// TIA Portal V19 export
FUNCTION "TRANSFER SUBOUTPUT" : Void   // FC13, LAD
{ S7_Optimized_Access := 'TRUE' }
// stored: SetENOAutomatically false
BEGIN

REGION Network 1: SYRUP MFG VESSEL BOTTOM STERROR RUN
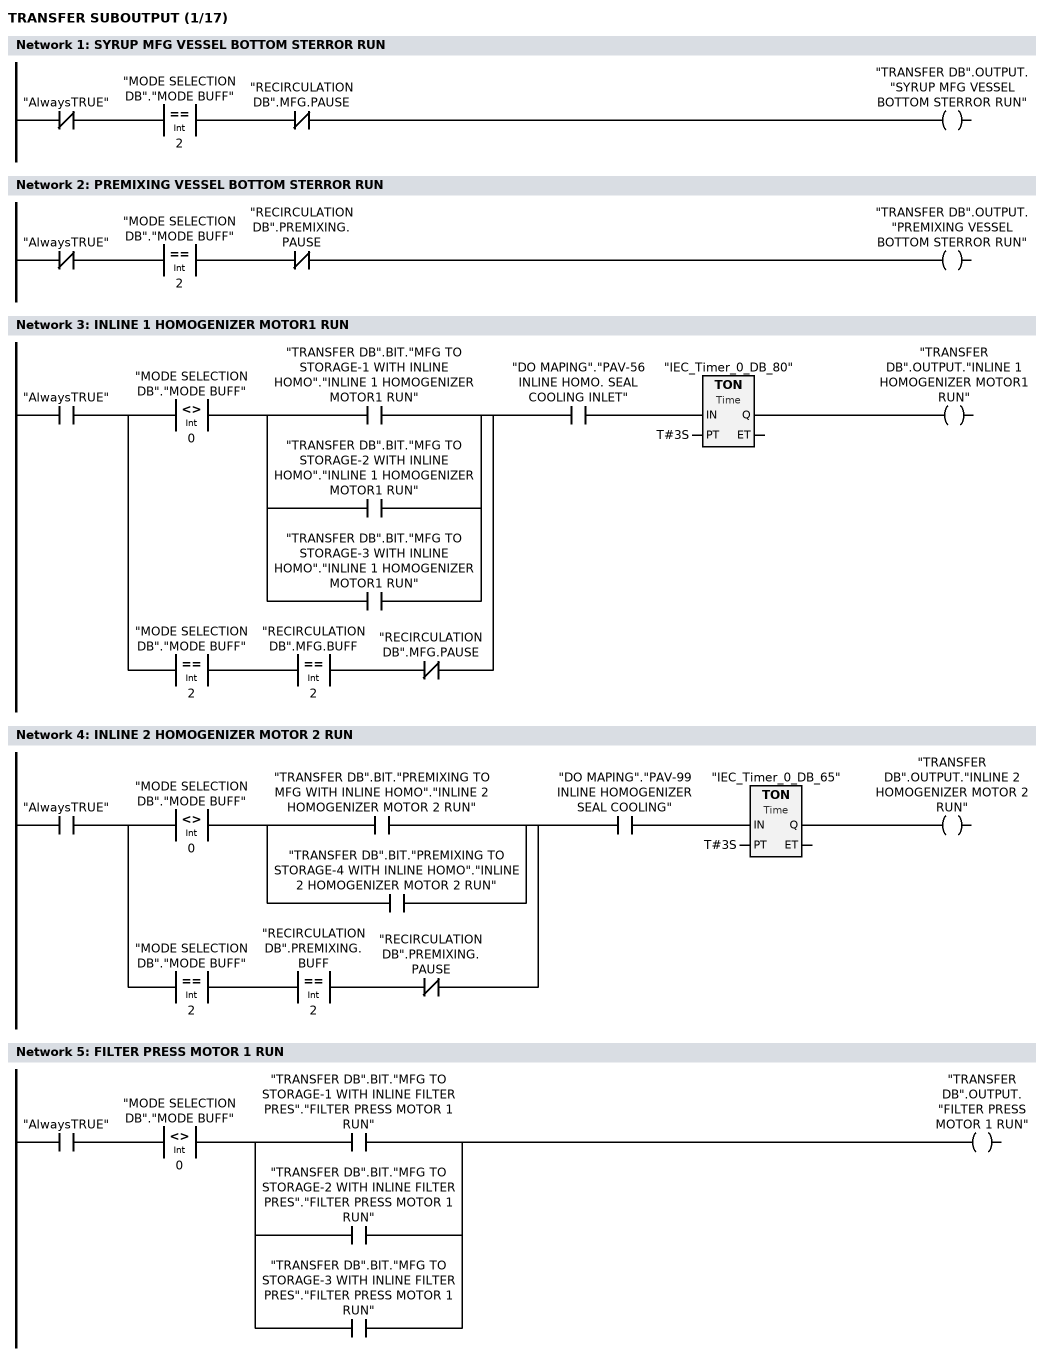
   RUNG wire#powerrail
      I_Contact( "AlwaysTRUE" )
      { S7_Templates := "SrcType := Int" } EQ_Contact(in1 := "MODE SELECTION DB"."MODE BUFF", in2 := 2)
      I_Contact( "RECIRCULATION DB".MFG.PAUSE )
      Coil( "TRANSFER DB".OUTPUT."SYRUP MFG VESSEL BOTTOM STERROR RUN" )
   END_RUNG
   // the same network as SCL:
   "TRANSFER DB".OUTPUT."SYRUP MFG VESSEL BOTTOM STERROR RUN" := NOT "AlwaysTRUE" AND ("MODE SELECTION DB"."MODE BUFF" = 2) AND NOT "RECIRCULATION DB".MFG.PAUSE;
END_REGION

REGION Network 2: PREMIXING VESSEL BOTTOM STERROR RUN
   RUNG wire#powerrail
      I_Contact( "AlwaysTRUE" )
      { S7_Templates := "SrcType := Int" } EQ_Contact(in1 := "MODE SELECTION DB"."MODE BUFF", in2 := 2)
      I_Contact( "RECIRCULATION DB".PREMIXING.PAUSE )
      Coil( "TRANSFER DB".OUTPUT."PREMIXING VESSEL BOTTOM STERROR RUN" )
   END_RUNG
   // the same network as SCL:
   "TRANSFER DB".OUTPUT."PREMIXING VESSEL BOTTOM STERROR RUN" := NOT "AlwaysTRUE" AND ("MODE SELECTION DB"."MODE BUFF" = 2) AND NOT "RECIRCULATION DB".PREMIXING.PAUSE;
END_REGION

REGION Network 3: INLINE 1 HOMOGENIZER MOTOR1 RUN
   RUNG wire#powerrail
      Contact( "AlwaysTRUE" )
      wire#w1
      { S7_Templates := "SrcType := Int" } NE_Contact(in1 := "MODE SELECTION DB"."MODE BUFF", in2 := 0)
      wire#w2
      Contact( "TRANSFER DB".BIT."MFG TO STORAGE-1 WITH INLINE HOMO"."INLINE 1 HOMOGENIZER MOTOR1 RUN" )
      wire#w3
      Contact( "DO MAPING"."PAV-56 INLINE HOMO. SEAL COOLING INLET" )
      { S7_Templates := "time_type := Time" } "IEC_Timer_0_DB_80".TON(pt := T#3S, et =>)
      Coil( "TRANSFER DB".OUTPUT."INLINE 1 HOMOGENIZER MOTOR1 RUN" )
   END_RUNG
   RUNG wire#w2
      Contact( "TRANSFER DB".BIT."MFG TO STORAGE-2 WITH INLINE HOMO"."INLINE 1 HOMOGENIZER MOTOR1 RUN" )
   END_RUNG wire#w3
   RUNG wire#w2
      Contact( "TRANSFER DB".BIT."MFG TO STORAGE-3 WITH INLINE HOMO"."INLINE 1 HOMOGENIZER MOTOR1 RUN" )
   END_RUNG wire#w3
   RUNG wire#w1
      { S7_Templates := "SrcType := Int" } EQ_Contact(in1 := "MODE SELECTION DB"."MODE BUFF", in2 := 2)
      { S7_Templates := "SrcType := Int" } EQ_Contact(in1 := "RECIRCULATION DB".MFG.BUFF, in2 := 2)
      I_Contact( "RECIRCULATION DB".MFG.PAUSE )
   END_RUNG wire#w3
   // the same network as SCL:
   "IEC_Timer_0_DB_80".TON(IN := "AlwaysTRUE" AND ((("MODE SELECTION DB"."MODE BUFF" <> 0) AND ("TRANSFER DB".BIT."MFG TO STORAGE-1 WITH INLINE HOMO"."INLINE 1 HOMOGENIZER MOTOR1 RUN" OR "TRANSFER DB".BIT."MFG TO STORAGE-2 WITH INLINE HOMO"."INLINE 1 HOMOGENIZER MOTOR1 RUN" OR "TRANSFER DB".BIT."MFG TO STORAGE-3 WITH INLINE HOMO"."INLINE 1 HOMOGENIZER MOTOR1 RUN")) OR (("MODE SELECTION DB"."MODE BUFF" = 2) AND ("RECIRCULATION DB".MFG.BUFF = 2) AND NOT "RECIRCULATION DB".MFG.PAUSE)) AND "DO MAPING"."PAV-56 INLINE HOMO. SEAL COOLING INLET",
                           PT := T#3S);
   "TRANSFER DB".OUTPUT."INLINE 1 HOMOGENIZER MOTOR1 RUN" := "IEC_Timer_0_DB_80".Q;
END_REGION

REGION Network 4: INLINE 2 HOMOGENIZER MOTOR 2 RUN
   RUNG wire#powerrail
      Contact( "AlwaysTRUE" )
      wire#w1
      { S7_Templates := "SrcType := Int" } NE_Contact(in1 := "MODE SELECTION DB"."MODE BUFF", in2 := 0)
      wire#w2
      Contact( "TRANSFER DB".BIT."PREMIXING TO MFG WITH INLINE HOMO"."INLINE 2 HOMOGENIZER MOTOR 2 RUN" )
      wire#w3
      Contact( "DO MAPING"."PAV-99 INLINE HOMOGENIZER SEAL COOLING" )
      { S7_Templates := "time_type := Time" } "IEC_Timer_0_DB_65".TON(pt := T#3S, et =>)
      Coil( "TRANSFER DB".OUTPUT."INLINE 2 HOMOGENIZER MOTOR 2 RUN" )
   END_RUNG
   RUNG wire#w2
      Contact( "TRANSFER DB".BIT."PREMIXING TO STORAGE-4 WITH INLINE HOMO"."INLINE 2 HOMOGENIZER MOTOR 2 RUN" )
   END_RUNG wire#w3
   RUNG wire#w1
      { S7_Templates := "SrcType := Int" } EQ_Contact(in1 := "MODE SELECTION DB"."MODE BUFF", in2 := 2)
      { S7_Templates := "SrcType := Int" } EQ_Contact(in1 := "RECIRCULATION DB".PREMIXING.BUFF, in2 := 2)
      I_Contact( "RECIRCULATION DB".PREMIXING.PAUSE )
   END_RUNG wire#w3
   // the same network as SCL:
   "IEC_Timer_0_DB_65".TON(IN := "AlwaysTRUE" AND ((("MODE SELECTION DB"."MODE BUFF" <> 0) AND ("TRANSFER DB".BIT."PREMIXING TO MFG WITH INLINE HOMO"."INLINE 2 HOMOGENIZER MOTOR 2 RUN" OR "TRANSFER DB".BIT."PREMIXING TO STORAGE-4 WITH INLINE HOMO"."INLINE 2 HOMOGENIZER MOTOR 2 RUN")) OR (("MODE SELECTION DB"."MODE BUFF" = 2) AND ("RECIRCULATION DB".PREMIXING.BUFF = 2) AND NOT "RECIRCULATION DB".PREMIXING.PAUSE)) AND "DO MAPING"."PAV-99 INLINE HOMOGENIZER SEAL COOLING",
                           PT := T#3S);
   "TRANSFER DB".OUTPUT."INLINE 2 HOMOGENIZER MOTOR 2 RUN" := "IEC_Timer_0_DB_65".Q;
END_REGION

REGION Network 5: FILTER PRESS MOTOR 1 RUN
   RUNG wire#powerrail
      Contact( "AlwaysTRUE" )
      { S7_Templates := "SrcType := Int" } NE_Contact(in1 := "MODE SELECTION DB"."MODE BUFF", in2 := 0)
      wire#w1
      Contact( "TRANSFER DB".BIT."MFG TO STORAGE-1 WITH INLINE FILTER PRES"."FILTER PRESS MOTOR 1 RUN" )
      wire#w2
      Coil( "TRANSFER DB".OUTPUT."FILTER PRESS MOTOR 1 RUN" )
   END_RUNG
   RUNG wire#w1
      Contact( "TRANSFER DB".BIT."MFG TO STORAGE-2 WITH INLINE FILTER PRES"."FILTER PRESS MOTOR 1 RUN" )
   END_RUNG wire#w2
   RUNG wire#w1
      Contact( "TRANSFER DB".BIT."MFG TO STORAGE-3 WITH INLINE FILTER PRES"."FILTER PRESS MOTOR 1 RUN" )
   END_RUNG wire#w2
   // the same network as SCL:
   "TRANSFER DB".OUTPUT."FILTER PRESS MOTOR 1 RUN" := "AlwaysTRUE" AND ("MODE SELECTION DB"."MODE BUFF" <> 0) AND ("TRANSFER DB".BIT."MFG TO STORAGE-1 WITH INLINE FILTER PRES"."FILTER PRESS MOTOR 1 RUN" OR "TRANSFER DB".BIT."MFG TO STORAGE-2 WITH INLINE FILTER PRES"."FILTER PRESS MOTOR 1 RUN" OR "TRANSFER DB".BIT."MFG TO STORAGE-3 WITH INLINE FILTER PRES"."FILTER PRESS MOTOR 1 RUN");
END_REGION

REGION Network 6: FILTER PRESS MOTOR 2 RUN
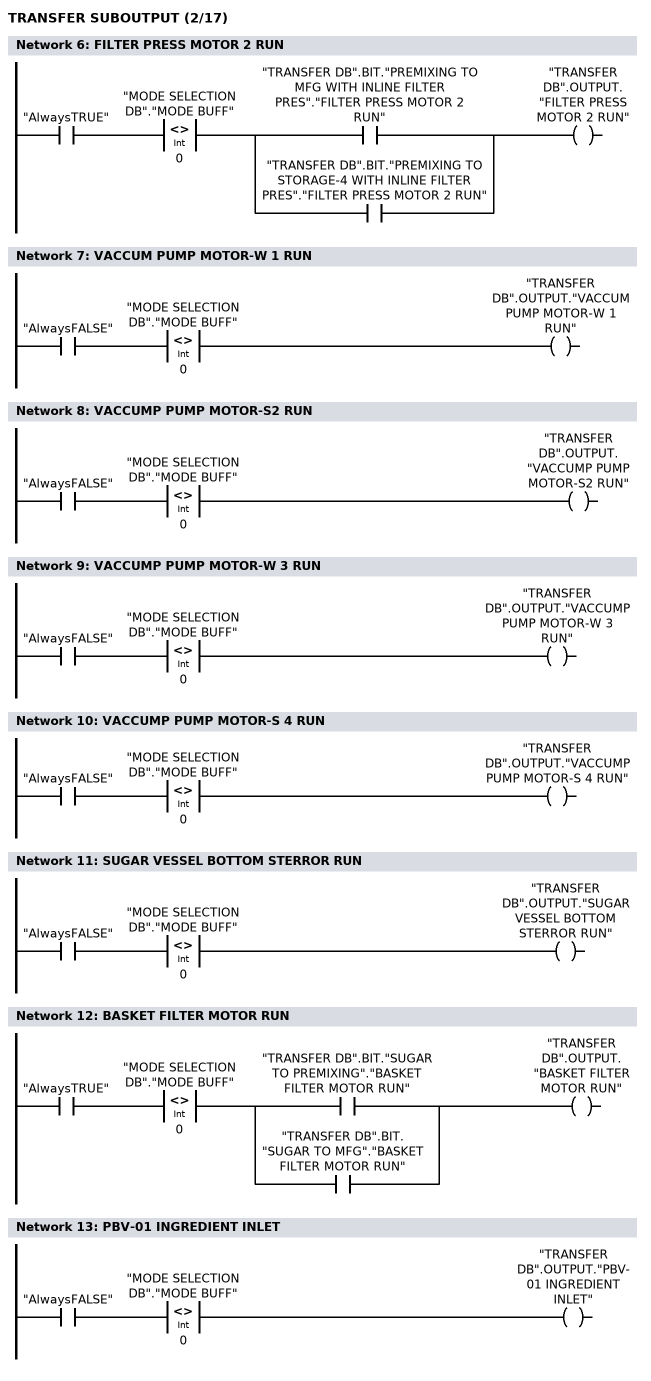
   RUNG wire#powerrail
      Contact( "AlwaysTRUE" )
      { S7_Templates := "SrcType := Int" } NE_Contact(in1 := "MODE SELECTION DB"."MODE BUFF", in2 := 0)
      wire#w1
      Contact( "TRANSFER DB".BIT."PREMIXING TO MFG WITH INLINE FILTER PRES"."FILTER PRESS MOTOR 2 RUN" )
      wire#w2
      Coil( "TRANSFER DB".OUTPUT."FILTER PRESS MOTOR 2 RUN" )
   END_RUNG
   RUNG wire#w1
      Contact( "TRANSFER DB".BIT."PREMIXING TO STORAGE-4 WITH INLINE FILTER PRES"."FILTER PRESS MOTOR 2 RUN" )
   END_RUNG wire#w2
   // the same network as SCL:
   "TRANSFER DB".OUTPUT."FILTER PRESS MOTOR 2 RUN" := "AlwaysTRUE" AND ("MODE SELECTION DB"."MODE BUFF" <> 0) AND ("TRANSFER DB".BIT."PREMIXING TO MFG WITH INLINE FILTER PRES"."FILTER PRESS MOTOR 2 RUN" OR "TRANSFER DB".BIT."PREMIXING TO STORAGE-4 WITH INLINE FILTER PRES"."FILTER PRESS MOTOR 2 RUN");
END_REGION

REGION Network 7: VACCUM PUMP MOTOR-W 1 RUN
   RUNG wire#powerrail
      Contact( "AlwaysFALSE" )
      { S7_Templates := "SrcType := Int" } NE_Contact(in1 := "MODE SELECTION DB"."MODE BUFF", in2 := 0)
      Coil( "TRANSFER DB".OUTPUT."VACCUM PUMP MOTOR-W 1 RUN" )
   END_RUNG
   // the same network as SCL:
   "TRANSFER DB".OUTPUT."VACCUM PUMP MOTOR-W 1 RUN" := "AlwaysFALSE" AND ("MODE SELECTION DB"."MODE BUFF" <> 0);
END_REGION

REGION Network 8: VACCUMP PUMP MOTOR-S2 RUN
   RUNG wire#powerrail
      Contact( "AlwaysFALSE" )
      { S7_Templates := "SrcType := Int" } NE_Contact(in1 := "MODE SELECTION DB"."MODE BUFF", in2 := 0)
      Coil( "TRANSFER DB".OUTPUT."VACCUMP PUMP MOTOR-S2 RUN" )
   END_RUNG
   // the same network as SCL:
   "TRANSFER DB".OUTPUT."VACCUMP PUMP MOTOR-S2 RUN" := "AlwaysFALSE" AND ("MODE SELECTION DB"."MODE BUFF" <> 0);
END_REGION

REGION Network 9: VACCUMP PUMP MOTOR-W 3 RUN
   RUNG wire#powerrail
      Contact( "AlwaysFALSE" )
      { S7_Templates := "SrcType := Int" } NE_Contact(in1 := "MODE SELECTION DB"."MODE BUFF", in2 := 0)
      Coil( "TRANSFER DB".OUTPUT."VACCUMP PUMP MOTOR-W 3 RUN" )
   END_RUNG
   // the same network as SCL:
   "TRANSFER DB".OUTPUT."VACCUMP PUMP MOTOR-W 3 RUN" := "AlwaysFALSE" AND ("MODE SELECTION DB"."MODE BUFF" <> 0);
END_REGION

REGION Network 10: VACCUMP PUMP MOTOR-S 4 RUN
   RUNG wire#powerrail
      Contact( "AlwaysFALSE" )
      { S7_Templates := "SrcType := Int" } NE_Contact(in1 := "MODE SELECTION DB"."MODE BUFF", in2 := 0)
      Coil( "TRANSFER DB".OUTPUT."VACCUMP PUMP MOTOR-S 4 RUN" )
   END_RUNG
   // the same network as SCL:
   "TRANSFER DB".OUTPUT."VACCUMP PUMP MOTOR-S 4 RUN" := "AlwaysFALSE" AND ("MODE SELECTION DB"."MODE BUFF" <> 0);
END_REGION

REGION Network 11: SUGAR VESSEL BOTTOM STERROR RUN
   RUNG wire#powerrail
      Contact( "AlwaysFALSE" )
      { S7_Templates := "SrcType := Int" } NE_Contact(in1 := "MODE SELECTION DB"."MODE BUFF", in2 := 0)
      Coil( "TRANSFER DB".OUTPUT."SUGAR VESSEL BOTTOM STERROR RUN" )
   END_RUNG
   // the same network as SCL:
   "TRANSFER DB".OUTPUT."SUGAR VESSEL BOTTOM STERROR RUN" := "AlwaysFALSE" AND ("MODE SELECTION DB"."MODE BUFF" <> 0);
END_REGION

REGION Network 12: BASKET FILTER MOTOR RUN
   RUNG wire#powerrail
      Contact( "AlwaysTRUE" )
      { S7_Templates := "SrcType := Int" } NE_Contact(in1 := "MODE SELECTION DB"."MODE BUFF", in2 := 0)
      wire#w1
      Contact( "TRANSFER DB".BIT."SUGAR TO PREMIXING"."BASKET FILTER MOTOR RUN" )
      wire#w2
      Coil( "TRANSFER DB".OUTPUT."BASKET FILTER MOTOR RUN" )
   END_RUNG
   RUNG wire#w1
      Contact( "TRANSFER DB".BIT."SUGAR TO MFG"."BASKET FILTER MOTOR RUN" )
   END_RUNG wire#w2
   // the same network as SCL:
   "TRANSFER DB".OUTPUT."BASKET FILTER MOTOR RUN" := "AlwaysTRUE" AND ("MODE SELECTION DB"."MODE BUFF" <> 0) AND ("TRANSFER DB".BIT."SUGAR TO PREMIXING"."BASKET FILTER MOTOR RUN" OR "TRANSFER DB".BIT."SUGAR TO MFG"."BASKET FILTER MOTOR RUN");
END_REGION

REGION Network 13: PBV-01 INGREDIENT INLET
   RUNG wire#powerrail
      Contact( "AlwaysFALSE" )
      { S7_Templates := "SrcType := Int" } NE_Contact(in1 := "MODE SELECTION DB"."MODE BUFF", in2 := 0)
      Coil( "TRANSFER DB".OUTPUT."PBV-01 INGREDIENT INLET" )
   END_RUNG
   // the same network as SCL:
   "TRANSFER DB".OUTPUT."PBV-01 INGREDIENT INLET" := "AlwaysFALSE" AND ("MODE SELECTION DB"."MODE BUFF" <> 0);
END_REGION

REGION Network 14: PBV-02 CIP INLET (SPRAY BALL)
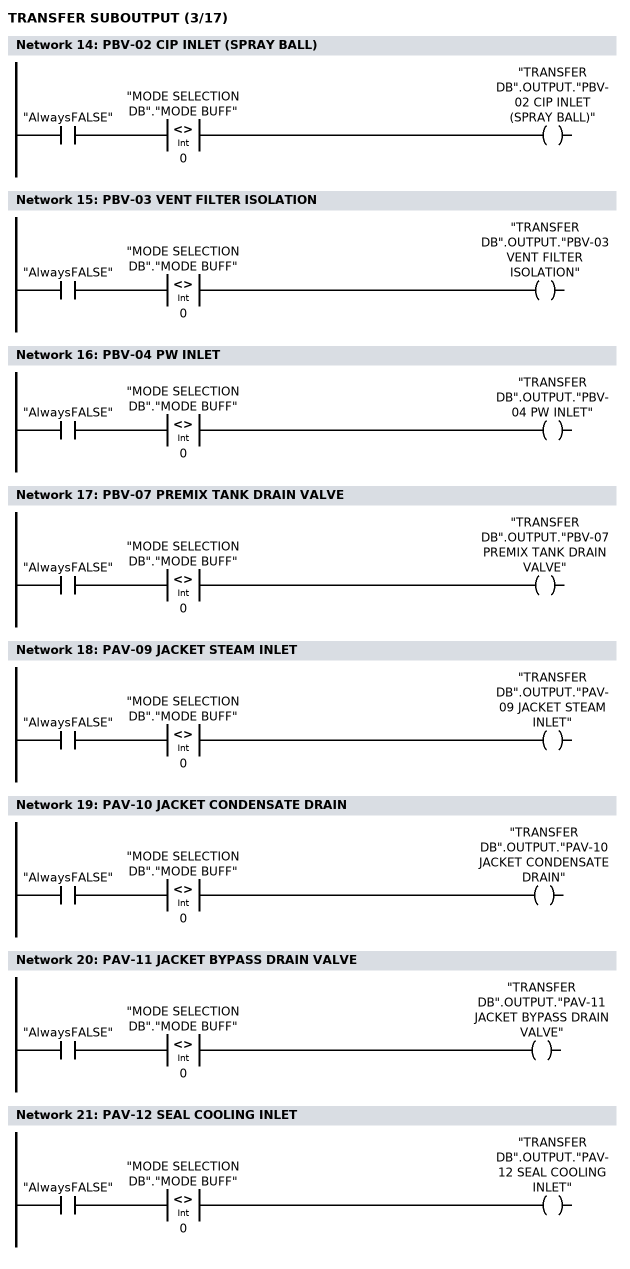
   RUNG wire#powerrail
      Contact( "AlwaysFALSE" )
      { S7_Templates := "SrcType := Int" } NE_Contact(in1 := "MODE SELECTION DB"."MODE BUFF", in2 := 0)
      Coil( "TRANSFER DB".OUTPUT."PBV-02 CIP INLET (SPRAY BALL)" )
   END_RUNG
   // the same network as SCL:
   "TRANSFER DB".OUTPUT."PBV-02 CIP INLET (SPRAY BALL)" := "AlwaysFALSE" AND ("MODE SELECTION DB"."MODE BUFF" <> 0);
END_REGION

REGION Network 15: PBV-03 VENT FILTER ISOLATION
   RUNG wire#powerrail
      Contact( "AlwaysFALSE" )
      { S7_Templates := "SrcType := Int" } NE_Contact(in1 := "MODE SELECTION DB"."MODE BUFF", in2 := 0)
      Coil( "TRANSFER DB".OUTPUT."PBV-03 VENT FILTER ISOLATION" )
   END_RUNG
   // the same network as SCL:
   "TRANSFER DB".OUTPUT."PBV-03 VENT FILTER ISOLATION" := "AlwaysFALSE" AND ("MODE SELECTION DB"."MODE BUFF" <> 0);
END_REGION

REGION Network 16: PBV-04 PW INLET
   RUNG wire#powerrail
      Contact( "AlwaysFALSE" )
      { S7_Templates := "SrcType := Int" } NE_Contact(in1 := "MODE SELECTION DB"."MODE BUFF", in2 := 0)
      Coil( "TRANSFER DB".OUTPUT."PBV-04 PW INLET" )
   END_RUNG
   // the same network as SCL:
   "TRANSFER DB".OUTPUT."PBV-04 PW INLET" := "AlwaysFALSE" AND ("MODE SELECTION DB"."MODE BUFF" <> 0);
END_REGION

REGION Network 17: PBV-07 PREMIX TANK DRAIN VALVE
   RUNG wire#powerrail
      Contact( "AlwaysFALSE" )
      { S7_Templates := "SrcType := Int" } NE_Contact(in1 := "MODE SELECTION DB"."MODE BUFF", in2 := 0)
      Coil( "TRANSFER DB".OUTPUT."PBV-07 PREMIX TANK DRAIN VALVE" )
   END_RUNG
   // the same network as SCL:
   "TRANSFER DB".OUTPUT."PBV-07 PREMIX TANK DRAIN VALVE" := "AlwaysFALSE" AND ("MODE SELECTION DB"."MODE BUFF" <> 0);
END_REGION

REGION Network 18: PAV-09 JACKET STEAM INLET
   RUNG wire#powerrail
      Contact( "AlwaysFALSE" )
      { S7_Templates := "SrcType := Int" } NE_Contact(in1 := "MODE SELECTION DB"."MODE BUFF", in2 := 0)
      Coil( "TRANSFER DB".OUTPUT."PAV-09 JACKET STEAM INLET" )
   END_RUNG
   // the same network as SCL:
   "TRANSFER DB".OUTPUT."PAV-09 JACKET STEAM INLET" := "AlwaysFALSE" AND ("MODE SELECTION DB"."MODE BUFF" <> 0);
END_REGION

REGION Network 19: PAV-10 JACKET CONDENSATE DRAIN
   RUNG wire#powerrail
      Contact( "AlwaysFALSE" )
      { S7_Templates := "SrcType := Int" } NE_Contact(in1 := "MODE SELECTION DB"."MODE BUFF", in2 := 0)
      Coil( "TRANSFER DB".OUTPUT."PAV-10 JACKET CONDENSATE DRAIN" )
   END_RUNG
   // the same network as SCL:
   "TRANSFER DB".OUTPUT."PAV-10 JACKET CONDENSATE DRAIN" := "AlwaysFALSE" AND ("MODE SELECTION DB"."MODE BUFF" <> 0);
END_REGION

REGION Network 20: PAV-11 JACKET BYPASS DRAIN VALVE
   RUNG wire#powerrail
      Contact( "AlwaysFALSE" )
      { S7_Templates := "SrcType := Int" } NE_Contact(in1 := "MODE SELECTION DB"."MODE BUFF", in2 := 0)
      Coil( "TRANSFER DB".OUTPUT."PAV-11 JACKET BYPASS DRAIN VALVE" )
   END_RUNG
   // the same network as SCL:
   "TRANSFER DB".OUTPUT."PAV-11 JACKET BYPASS DRAIN VALVE" := "AlwaysFALSE" AND ("MODE SELECTION DB"."MODE BUFF" <> 0);
END_REGION

REGION Network 21: PAV-12 SEAL COOLING INLET
   RUNG wire#powerrail
      Contact( "AlwaysFALSE" )
      { S7_Templates := "SrcType := Int" } NE_Contact(in1 := "MODE SELECTION DB"."MODE BUFF", in2 := 0)
      Coil( "TRANSFER DB".OUTPUT."PAV-12 SEAL COOLING INLET" )
   END_RUNG
   // the same network as SCL:
   "TRANSFER DB".OUTPUT."PAV-12 SEAL COOLING INLET" := "AlwaysFALSE" AND ("MODE SELECTION DB"."MODE BUFF" <> 0);
END_REGION

REGION Network 22: PAV-13 WATER COOLING INLET
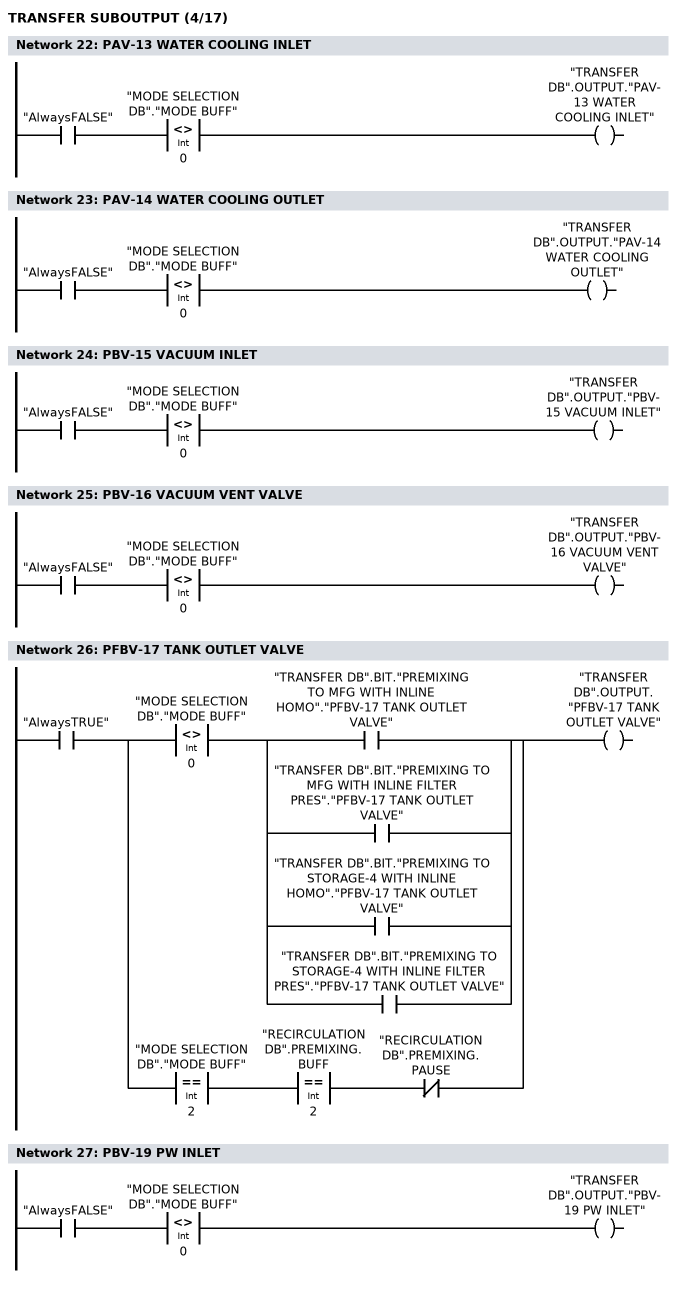
   RUNG wire#powerrail
      Contact( "AlwaysFALSE" )
      { S7_Templates := "SrcType := Int" } NE_Contact(in1 := "MODE SELECTION DB"."MODE BUFF", in2 := 0)
      Coil( "TRANSFER DB".OUTPUT."PAV-13 WATER COOLING INLET" )
   END_RUNG
   // the same network as SCL:
   "TRANSFER DB".OUTPUT."PAV-13 WATER COOLING INLET" := "AlwaysFALSE" AND ("MODE SELECTION DB"."MODE BUFF" <> 0);
END_REGION

REGION Network 23: PAV-14 WATER COOLING OUTLET
   RUNG wire#powerrail
      Contact( "AlwaysFALSE" )
      { S7_Templates := "SrcType := Int" } NE_Contact(in1 := "MODE SELECTION DB"."MODE BUFF", in2 := 0)
      Coil( "TRANSFER DB".OUTPUT."PAV-14 WATER COOLING OUTLET" )
   END_RUNG
   // the same network as SCL:
   "TRANSFER DB".OUTPUT."PAV-14 WATER COOLING OUTLET" := "AlwaysFALSE" AND ("MODE SELECTION DB"."MODE BUFF" <> 0);
END_REGION

REGION Network 24: PBV-15 VACUUM INLET
   RUNG wire#powerrail
      Contact( "AlwaysFALSE" )
      { S7_Templates := "SrcType := Int" } NE_Contact(in1 := "MODE SELECTION DB"."MODE BUFF", in2 := 0)
      Coil( "TRANSFER DB".OUTPUT."PBV-15 VACUUM INLET" )
   END_RUNG
   // the same network as SCL:
   "TRANSFER DB".OUTPUT."PBV-15 VACUUM INLET" := "AlwaysFALSE" AND ("MODE SELECTION DB"."MODE BUFF" <> 0);
END_REGION

REGION Network 25: PBV-16 VACUUM VENT VALVE
   RUNG wire#powerrail
      Contact( "AlwaysFALSE" )
      { S7_Templates := "SrcType := Int" } NE_Contact(in1 := "MODE SELECTION DB"."MODE BUFF", in2 := 0)
      Coil( "TRANSFER DB".OUTPUT."PBV-16 VACUUM VENT VALVE" )
   END_RUNG
   // the same network as SCL:
   "TRANSFER DB".OUTPUT."PBV-16 VACUUM VENT VALVE" := "AlwaysFALSE" AND ("MODE SELECTION DB"."MODE BUFF" <> 0);
END_REGION

REGION Network 26: PFBV-17 TANK OUTLET VALVE
   RUNG wire#powerrail
      Contact( "AlwaysTRUE" )
      wire#w1
      { S7_Templates := "SrcType := Int" } NE_Contact(in1 := "MODE SELECTION DB"."MODE BUFF", in2 := 0)
      wire#w2
      Contact( "TRANSFER DB".BIT."PREMIXING TO MFG WITH INLINE HOMO"."PFBV-17 TANK OUTLET VALVE" )
      wire#w3
      Coil( "TRANSFER DB".OUTPUT."PFBV-17 TANK OUTLET VALVE" )
   END_RUNG
   RUNG wire#w2
      Contact( "TRANSFER DB".BIT."PREMIXING TO MFG WITH INLINE FILTER PRES"."PFBV-17 TANK OUTLET VALVE" )
   END_RUNG wire#w3
   RUNG wire#w2
      Contact( "TRANSFER DB".BIT."PREMIXING TO STORAGE-4 WITH INLINE HOMO"."PFBV-17 TANK OUTLET VALVE" )
   END_RUNG wire#w3
   RUNG wire#w2
      Contact( "TRANSFER DB".BIT."PREMIXING TO STORAGE-4 WITH INLINE FILTER PRES"."PFBV-17 TANK OUTLET VALVE" )
   END_RUNG wire#w3
   RUNG wire#w1
      { S7_Templates := "SrcType := Int" } EQ_Contact(in1 := "MODE SELECTION DB"."MODE BUFF", in2 := 2)
      { S7_Templates := "SrcType := Int" } EQ_Contact(in1 := "RECIRCULATION DB".PREMIXING.BUFF, in2 := 2)
      I_Contact( "RECIRCULATION DB".PREMIXING.PAUSE )
   END_RUNG wire#w3
   // the same network as SCL:
   "TRANSFER DB".OUTPUT."PFBV-17 TANK OUTLET VALVE" := "AlwaysTRUE" AND ((("MODE SELECTION DB"."MODE BUFF" <> 0) AND ("TRANSFER DB".BIT."PREMIXING TO MFG WITH INLINE HOMO"."PFBV-17 TANK OUTLET VALVE" OR "TRANSFER DB".BIT."PREMIXING TO MFG WITH INLINE FILTER PRES"."PFBV-17 TANK OUTLET VALVE" OR "TRANSFER DB".BIT."PREMIXING TO STORAGE-4 WITH INLINE HOMO"."PFBV-17 TANK OUTLET VALVE" OR "TRANSFER DB".BIT."PREMIXING TO STORAGE-4 WITH INLINE FILTER PRES"."PFBV-17 TANK OUTLET VALVE")) OR (("MODE SELECTION DB"."MODE BUFF" = 2) AND ("RECIRCULATION DB".PREMIXING.BUFF = 2) AND NOT "RECIRCULATION DB".PREMIXING.PAUSE));
END_REGION

REGION Network 27: PBV-19 PW INLET
   RUNG wire#powerrail
      Contact( "AlwaysFALSE" )
      { S7_Templates := "SrcType := Int" } NE_Contact(in1 := "MODE SELECTION DB"."MODE BUFF", in2 := 0)
      Coil( "TRANSFER DB".OUTPUT."PBV-19 PW INLET" )
   END_RUNG
   // the same network as SCL:
   "TRANSFER DB".OUTPUT."PBV-19 PW INLET" := "AlwaysFALSE" AND ("MODE SELECTION DB"."MODE BUFF" <> 0);
END_REGION

REGION Network 28: PBV-20 CIP INLET (SPRAY BALL)
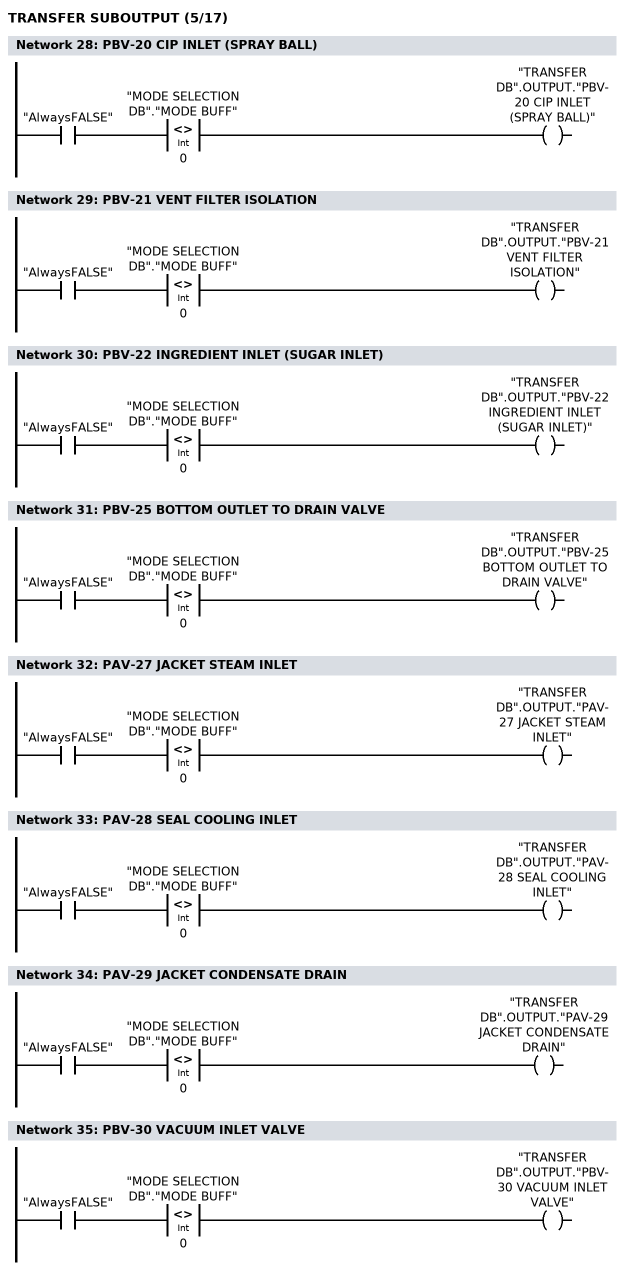
   RUNG wire#powerrail
      Contact( "AlwaysFALSE" )
      { S7_Templates := "SrcType := Int" } NE_Contact(in1 := "MODE SELECTION DB"."MODE BUFF", in2 := 0)
      Coil( "TRANSFER DB".OUTPUT."PBV-20 CIP INLET (SPRAY BALL)" )
   END_RUNG
   // the same network as SCL:
   "TRANSFER DB".OUTPUT."PBV-20 CIP INLET (SPRAY BALL)" := "AlwaysFALSE" AND ("MODE SELECTION DB"."MODE BUFF" <> 0);
END_REGION

REGION Network 29: PBV-21 VENT FILTER ISOLATION
   RUNG wire#powerrail
      Contact( "AlwaysFALSE" )
      { S7_Templates := "SrcType := Int" } NE_Contact(in1 := "MODE SELECTION DB"."MODE BUFF", in2 := 0)
      Coil( "TRANSFER DB".OUTPUT."PBV-21 VENT FILTER ISOLATION" )
   END_RUNG
   // the same network as SCL:
   "TRANSFER DB".OUTPUT."PBV-21 VENT FILTER ISOLATION" := "AlwaysFALSE" AND ("MODE SELECTION DB"."MODE BUFF" <> 0);
END_REGION

REGION Network 30: PBV-22 INGREDIENT INLET (SUGAR INLET)
   RUNG wire#powerrail
      Contact( "AlwaysFALSE" )
      { S7_Templates := "SrcType := Int" } NE_Contact(in1 := "MODE SELECTION DB"."MODE BUFF", in2 := 0)
      Coil( "TRANSFER DB".OUTPUT."PBV-22 INGREDIENT INLET (SUGAR INLET)" )
   END_RUNG
   // the same network as SCL:
   "TRANSFER DB".OUTPUT."PBV-22 INGREDIENT INLET (SUGAR INLET)" := "AlwaysFALSE" AND ("MODE SELECTION DB"."MODE BUFF" <> 0);
END_REGION

REGION Network 31: PBV-25 BOTTOM OUTLET TO DRAIN VALVE
   RUNG wire#powerrail
      Contact( "AlwaysFALSE" )
      { S7_Templates := "SrcType := Int" } NE_Contact(in1 := "MODE SELECTION DB"."MODE BUFF", in2 := 0)
      Coil( "TRANSFER DB".OUTPUT."PBV-25 BOTTOM OUTLET TO DRAIN VALVE" )
   END_RUNG
   // the same network as SCL:
   "TRANSFER DB".OUTPUT."PBV-25 BOTTOM OUTLET TO DRAIN VALVE" := "AlwaysFALSE" AND ("MODE SELECTION DB"."MODE BUFF" <> 0);
END_REGION

REGION Network 32: PAV-27 JACKET STEAM INLET
   RUNG wire#powerrail
      Contact( "AlwaysFALSE" )
      { S7_Templates := "SrcType := Int" } NE_Contact(in1 := "MODE SELECTION DB"."MODE BUFF", in2 := 0)
      Coil( "TRANSFER DB".OUTPUT."PAV-27 JACKET STEAM INLET" )
   END_RUNG
   // the same network as SCL:
   "TRANSFER DB".OUTPUT."PAV-27 JACKET STEAM INLET" := "AlwaysFALSE" AND ("MODE SELECTION DB"."MODE BUFF" <> 0);
END_REGION

REGION Network 33: PAV-28 SEAL COOLING INLET
   RUNG wire#powerrail
      Contact( "AlwaysFALSE" )
      { S7_Templates := "SrcType := Int" } NE_Contact(in1 := "MODE SELECTION DB"."MODE BUFF", in2 := 0)
      Coil( "TRANSFER DB".OUTPUT."PAV-28 SEAL COOLING INLET" )
   END_RUNG
   // the same network as SCL:
   "TRANSFER DB".OUTPUT."PAV-28 SEAL COOLING INLET" := "AlwaysFALSE" AND ("MODE SELECTION DB"."MODE BUFF" <> 0);
END_REGION

REGION Network 34: PAV-29 JACKET CONDENSATE DRAIN
   RUNG wire#powerrail
      Contact( "AlwaysFALSE" )
      { S7_Templates := "SrcType := Int" } NE_Contact(in1 := "MODE SELECTION DB"."MODE BUFF", in2 := 0)
      Coil( "TRANSFER DB".OUTPUT."PAV-29 JACKET CONDENSATE DRAIN" )
   END_RUNG
   // the same network as SCL:
   "TRANSFER DB".OUTPUT."PAV-29 JACKET CONDENSATE DRAIN" := "AlwaysFALSE" AND ("MODE SELECTION DB"."MODE BUFF" <> 0);
END_REGION

REGION Network 35: PBV-30 VACUUM INLET VALVE
   RUNG wire#powerrail
      Contact( "AlwaysFALSE" )
      { S7_Templates := "SrcType := Int" } NE_Contact(in1 := "MODE SELECTION DB"."MODE BUFF", in2 := 0)
      Coil( "TRANSFER DB".OUTPUT."PBV-30 VACUUM INLET VALVE" )
   END_RUNG
   // the same network as SCL:
   "TRANSFER DB".OUTPUT."PBV-30 VACUUM INLET VALVE" := "AlwaysFALSE" AND ("MODE SELECTION DB"."MODE BUFF" <> 0);
END_REGION

REGION Network 36: PBV-31 VACUUM VENT VALVE
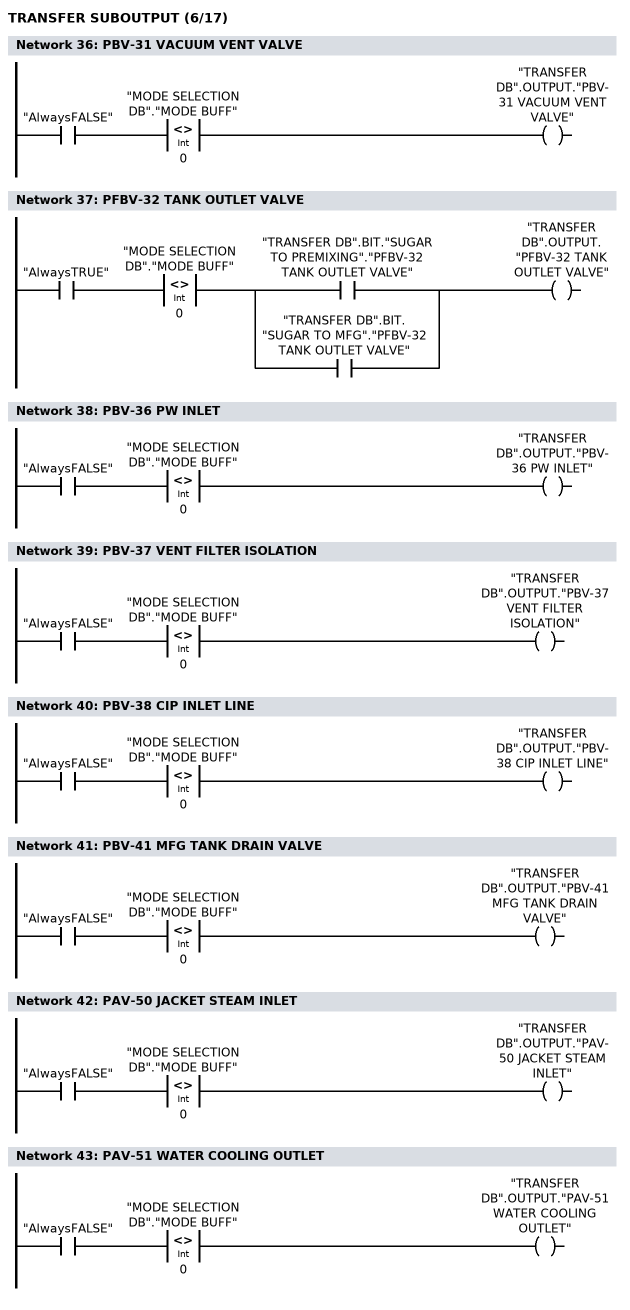
   RUNG wire#powerrail
      Contact( "AlwaysFALSE" )
      { S7_Templates := "SrcType := Int" } NE_Contact(in1 := "MODE SELECTION DB"."MODE BUFF", in2 := 0)
      Coil( "TRANSFER DB".OUTPUT."PBV-31 VACUUM VENT VALVE" )
   END_RUNG
   // the same network as SCL:
   "TRANSFER DB".OUTPUT."PBV-31 VACUUM VENT VALVE" := "AlwaysFALSE" AND ("MODE SELECTION DB"."MODE BUFF" <> 0);
END_REGION

REGION Network 37: PFBV-32 TANK OUTLET VALVE
   RUNG wire#powerrail
      Contact( "AlwaysTRUE" )
      { S7_Templates := "SrcType := Int" } NE_Contact(in1 := "MODE SELECTION DB"."MODE BUFF", in2 := 0)
      wire#w1
      Contact( "TRANSFER DB".BIT."SUGAR TO PREMIXING"."PFBV-32 TANK OUTLET VALVE" )
      wire#w2
      Coil( "TRANSFER DB".OUTPUT."PFBV-32 TANK OUTLET VALVE" )
   END_RUNG
   RUNG wire#w1
      Contact( "TRANSFER DB".BIT."SUGAR TO MFG"."PFBV-32 TANK OUTLET VALVE" )
   END_RUNG wire#w2
   // the same network as SCL:
   "TRANSFER DB".OUTPUT."PFBV-32 TANK OUTLET VALVE" := "AlwaysTRUE" AND ("MODE SELECTION DB"."MODE BUFF" <> 0) AND ("TRANSFER DB".BIT."SUGAR TO PREMIXING"."PFBV-32 TANK OUTLET VALVE" OR "TRANSFER DB".BIT."SUGAR TO MFG"."PFBV-32 TANK OUTLET VALVE");
END_REGION

REGION Network 38: PBV-36 PW INLET
   RUNG wire#powerrail
      Contact( "AlwaysFALSE" )
      { S7_Templates := "SrcType := Int" } NE_Contact(in1 := "MODE SELECTION DB"."MODE BUFF", in2 := 0)
      Coil( "TRANSFER DB".OUTPUT."PBV-36 PW INLET" )
   END_RUNG
   // the same network as SCL:
   "TRANSFER DB".OUTPUT."PBV-36 PW INLET" := "AlwaysFALSE" AND ("MODE SELECTION DB"."MODE BUFF" <> 0);
END_REGION

REGION Network 39: PBV-37 VENT FILTER ISOLATION
   RUNG wire#powerrail
      Contact( "AlwaysFALSE" )
      { S7_Templates := "SrcType := Int" } NE_Contact(in1 := "MODE SELECTION DB"."MODE BUFF", in2 := 0)
      Coil( "TRANSFER DB".OUTPUT."PBV-37 VENT FILTER ISOLATION" )
   END_RUNG
   // the same network as SCL:
   "TRANSFER DB".OUTPUT."PBV-37 VENT FILTER ISOLATION" := "AlwaysFALSE" AND ("MODE SELECTION DB"."MODE BUFF" <> 0);
END_REGION

REGION Network 40: PBV-38 CIP INLET LINE
   RUNG wire#powerrail
      Contact( "AlwaysFALSE" )
      { S7_Templates := "SrcType := Int" } NE_Contact(in1 := "MODE SELECTION DB"."MODE BUFF", in2 := 0)
      Coil( "TRANSFER DB".OUTPUT."PBV-38 CIP INLET LINE" )
   END_RUNG
   // the same network as SCL:
   "TRANSFER DB".OUTPUT."PBV-38 CIP INLET LINE" := "AlwaysFALSE" AND ("MODE SELECTION DB"."MODE BUFF" <> 0);
END_REGION

REGION Network 41: PBV-41 MFG TANK DRAIN VALVE
   RUNG wire#powerrail
      Contact( "AlwaysFALSE" )
      { S7_Templates := "SrcType := Int" } NE_Contact(in1 := "MODE SELECTION DB"."MODE BUFF", in2 := 0)
      Coil( "TRANSFER DB".OUTPUT."PBV-41 MFG TANK DRAIN VALVE" )
   END_RUNG
   // the same network as SCL:
   "TRANSFER DB".OUTPUT."PBV-41 MFG TANK DRAIN VALVE" := "AlwaysFALSE" AND ("MODE SELECTION DB"."MODE BUFF" <> 0);
END_REGION

REGION Network 42: PAV-50 JACKET STEAM INLET
   RUNG wire#powerrail
      Contact( "AlwaysFALSE" )
      { S7_Templates := "SrcType := Int" } NE_Contact(in1 := "MODE SELECTION DB"."MODE BUFF", in2 := 0)
      Coil( "TRANSFER DB".OUTPUT."PAV-50 JACKET STEAM INLET" )
   END_RUNG
   // the same network as SCL:
   "TRANSFER DB".OUTPUT."PAV-50 JACKET STEAM INLET" := "AlwaysFALSE" AND ("MODE SELECTION DB"."MODE BUFF" <> 0);
END_REGION

REGION Network 43: PAV-51 WATER COOLING OUTLET
   RUNG wire#powerrail
      Contact( "AlwaysFALSE" )
      { S7_Templates := "SrcType := Int" } NE_Contact(in1 := "MODE SELECTION DB"."MODE BUFF", in2 := 0)
      Coil( "TRANSFER DB".OUTPUT."PAV-51 WATER COOLING OUTLET" )
   END_RUNG
   // the same network as SCL:
   "TRANSFER DB".OUTPUT."PAV-51 WATER COOLING OUTLET" := "AlwaysFALSE" AND ("MODE SELECTION DB"."MODE BUFF" <> 0);
END_REGION

REGION Network 44: PAV-52 WATER COOLING INLET
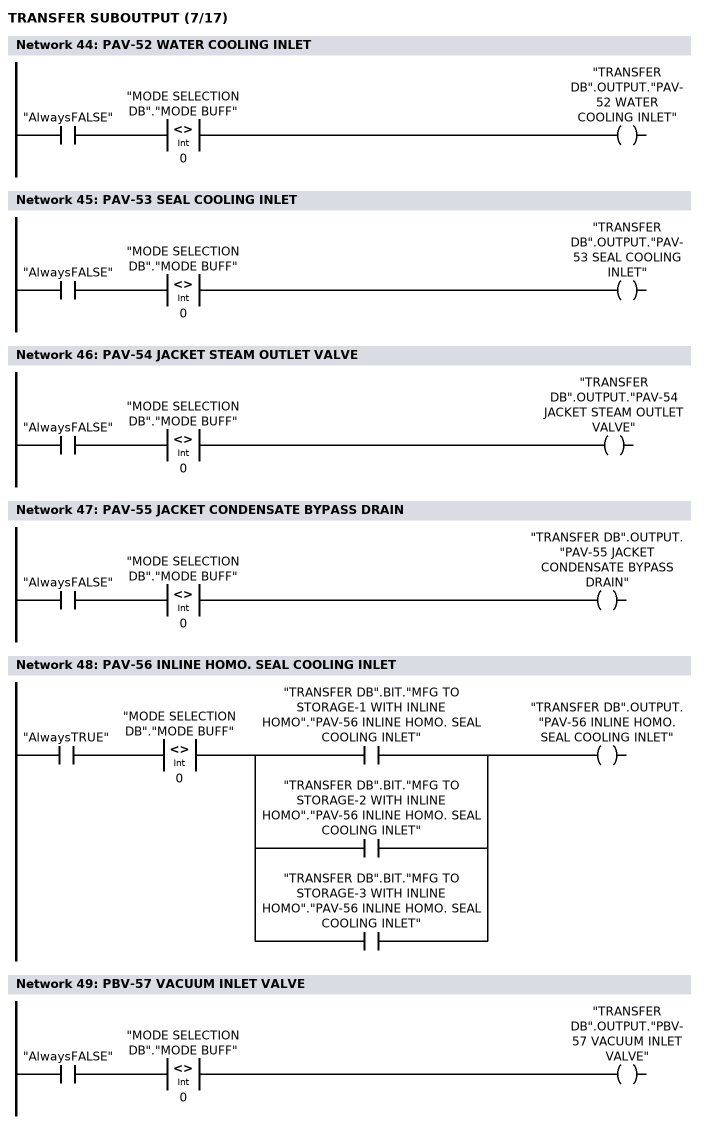
   RUNG wire#powerrail
      Contact( "AlwaysFALSE" )
      { S7_Templates := "SrcType := Int" } NE_Contact(in1 := "MODE SELECTION DB"."MODE BUFF", in2 := 0)
      Coil( "TRANSFER DB".OUTPUT."PAV-52 WATER COOLING INLET" )
   END_RUNG
   // the same network as SCL:
   "TRANSFER DB".OUTPUT."PAV-52 WATER COOLING INLET" := "AlwaysFALSE" AND ("MODE SELECTION DB"."MODE BUFF" <> 0);
END_REGION

REGION Network 45: PAV-53 SEAL COOLING INLET
   RUNG wire#powerrail
      Contact( "AlwaysFALSE" )
      { S7_Templates := "SrcType := Int" } NE_Contact(in1 := "MODE SELECTION DB"."MODE BUFF", in2 := 0)
      Coil( "TRANSFER DB".OUTPUT."PAV-53 SEAL COOLING INLET" )
   END_RUNG
   // the same network as SCL:
   "TRANSFER DB".OUTPUT."PAV-53 SEAL COOLING INLET" := "AlwaysFALSE" AND ("MODE SELECTION DB"."MODE BUFF" <> 0);
END_REGION

REGION Network 46: PAV-54 JACKET STEAM OUTLET VALVE
   RUNG wire#powerrail
      Contact( "AlwaysFALSE" )
      { S7_Templates := "SrcType := Int" } NE_Contact(in1 := "MODE SELECTION DB"."MODE BUFF", in2 := 0)
      Coil( "TRANSFER DB".OUTPUT."PAV-54 JACKET STEAM OUTLET VALVE" )
   END_RUNG
   // the same network as SCL:
   "TRANSFER DB".OUTPUT."PAV-54 JACKET STEAM OUTLET VALVE" := "AlwaysFALSE" AND ("MODE SELECTION DB"."MODE BUFF" <> 0);
END_REGION

REGION Network 47: PAV-55 JACKET CONDENSATE BYPASS DRAIN
   RUNG wire#powerrail
      Contact( "AlwaysFALSE" )
      { S7_Templates := "SrcType := Int" } NE_Contact(in1 := "MODE SELECTION DB"."MODE BUFF", in2 := 0)
      Coil( "TRANSFER DB".OUTPUT."PAV-55 JACKET CONDENSATE BYPASS DRAIN" )
   END_RUNG
   // the same network as SCL:
   "TRANSFER DB".OUTPUT."PAV-55 JACKET CONDENSATE BYPASS DRAIN" := "AlwaysFALSE" AND ("MODE SELECTION DB"."MODE BUFF" <> 0);
END_REGION

REGION Network 48: PAV-56 INLINE HOMO. SEAL COOLING INLET
   RUNG wire#powerrail
      Contact( "AlwaysTRUE" )
      { S7_Templates := "SrcType := Int" } NE_Contact(in1 := "MODE SELECTION DB"."MODE BUFF", in2 := 0)
      wire#w1
      Contact( "TRANSFER DB".BIT."MFG TO STORAGE-1 WITH INLINE HOMO"."PAV-56 INLINE HOMO. SEAL COOLING INLET" )
      wire#w2
      Coil( "TRANSFER DB".OUTPUT."PAV-56 INLINE HOMO. SEAL COOLING INLET" )
   END_RUNG
   RUNG wire#w1
      Contact( "TRANSFER DB".BIT."MFG TO STORAGE-2 WITH INLINE HOMO"."PAV-56 INLINE HOMO. SEAL COOLING INLET" )
   END_RUNG wire#w2
   RUNG wire#w1
      Contact( "TRANSFER DB".BIT."MFG TO STORAGE-3 WITH INLINE HOMO"."PAV-56 INLINE HOMO. SEAL COOLING INLET" )
   END_RUNG wire#w2
   // the same network as SCL:
   "TRANSFER DB".OUTPUT."PAV-56 INLINE HOMO. SEAL COOLING INLET" := "AlwaysTRUE" AND ("MODE SELECTION DB"."MODE BUFF" <> 0) AND ("TRANSFER DB".BIT."MFG TO STORAGE-1 WITH INLINE HOMO"."PAV-56 INLINE HOMO. SEAL COOLING INLET" OR "TRANSFER DB".BIT."MFG TO STORAGE-2 WITH INLINE HOMO"."PAV-56 INLINE HOMO. SEAL COOLING INLET" OR "TRANSFER DB".BIT."MFG TO STORAGE-3 WITH INLINE HOMO"."PAV-56 INLINE HOMO. SEAL COOLING INLET");
END_REGION

REGION Network 49: PBV-57 VACUUM INLET VALVE
   RUNG wire#powerrail
      Contact( "AlwaysFALSE" )
      { S7_Templates := "SrcType := Int" } NE_Contact(in1 := "MODE SELECTION DB"."MODE BUFF", in2 := 0)
      Coil( "TRANSFER DB".OUTPUT."PBV-57 VACUUM INLET VALVE" )
   END_RUNG
   // the same network as SCL:
   "TRANSFER DB".OUTPUT."PBV-57 VACUUM INLET VALVE" := "AlwaysFALSE" AND ("MODE SELECTION DB"."MODE BUFF" <> 0);
END_REGION

REGION Network 50: PFBV-59 TANK OUTLET VALVE
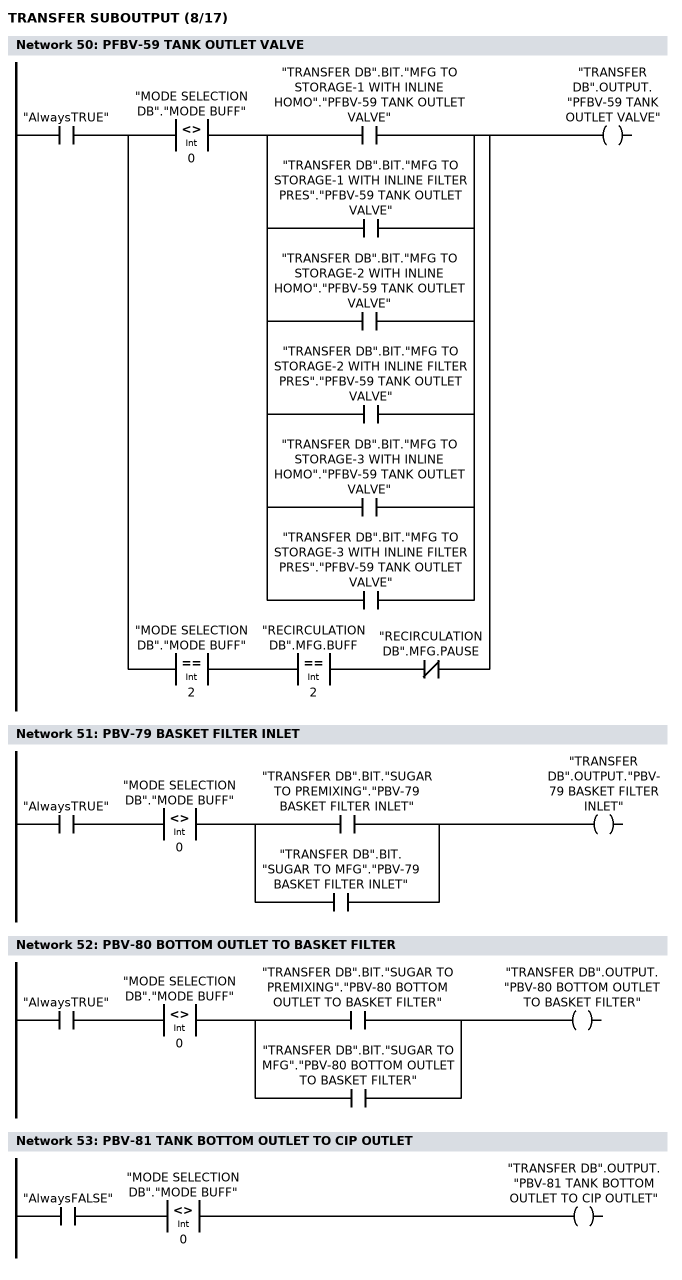
   RUNG wire#powerrail
      Contact( "AlwaysTRUE" )
      wire#w1
      { S7_Templates := "SrcType := Int" } NE_Contact(in1 := "MODE SELECTION DB"."MODE BUFF", in2 := 0)
      wire#w2
      Contact( "TRANSFER DB".BIT."MFG TO STORAGE-1 WITH INLINE HOMO"."PFBV-59 TANK OUTLET VALVE" )
      wire#w3
      Coil( "TRANSFER DB".OUTPUT."PFBV-59 TANK OUTLET VALVE" )
   END_RUNG
   RUNG wire#w2
      Contact( "TRANSFER DB".BIT."MFG TO STORAGE-1 WITH INLINE FILTER PRES"."PFBV-59 TANK OUTLET VALVE" )
   END_RUNG wire#w3
   RUNG wire#w2
      Contact( "TRANSFER DB".BIT."MFG TO STORAGE-2 WITH INLINE HOMO"."PFBV-59 TANK OUTLET VALVE" )
   END_RUNG wire#w3
   RUNG wire#w2
      Contact( "TRANSFER DB".BIT."MFG TO STORAGE-2 WITH INLINE FILTER PRES"."PFBV-59 TANK OUTLET VALVE" )
   END_RUNG wire#w3
   RUNG wire#w2
      Contact( "TRANSFER DB".BIT."MFG TO STORAGE-3 WITH INLINE HOMO"."PFBV-59 TANK OUTLET VALVE" )
   END_RUNG wire#w3
   RUNG wire#w2
      Contact( "TRANSFER DB".BIT."MFG TO STORAGE-3 WITH INLINE FILTER PRES"."PFBV-59 TANK OUTLET VALVE" )
   END_RUNG wire#w3
   RUNG wire#w1
      { S7_Templates := "SrcType := Int" } EQ_Contact(in1 := "MODE SELECTION DB"."MODE BUFF", in2 := 2)
      { S7_Templates := "SrcType := Int" } EQ_Contact(in1 := "RECIRCULATION DB".MFG.BUFF, in2 := 2)
      I_Contact( "RECIRCULATION DB".MFG.PAUSE )
   END_RUNG wire#w3
   // the same network as SCL:
   "TRANSFER DB".OUTPUT."PFBV-59 TANK OUTLET VALVE" := "AlwaysTRUE" AND ((("MODE SELECTION DB"."MODE BUFF" <> 0) AND ("TRANSFER DB".BIT."MFG TO STORAGE-1 WITH INLINE HOMO"."PFBV-59 TANK OUTLET VALVE" OR "TRANSFER DB".BIT."MFG TO STORAGE-1 WITH INLINE FILTER PRES"."PFBV-59 TANK OUTLET VALVE" OR "TRANSFER DB".BIT."MFG TO STORAGE-2 WITH INLINE HOMO"."PFBV-59 TANK OUTLET VALVE" OR "TRANSFER DB".BIT."MFG TO STORAGE-2 WITH INLINE FILTER PRES"."PFBV-59 TANK OUTLET VALVE" OR "TRANSFER DB".BIT."MFG TO STORAGE-3 WITH INLINE HOMO"."PFBV-59 TANK OUTLET VALVE" OR "TRANSFER DB".BIT."MFG TO STORAGE-3 WITH INLINE FILTER PRES"."PFBV-59 TANK OUTLET VALVE")) OR (("MODE SELECTION DB"."MODE BUFF" = 2) AND ("RECIRCULATION DB".MFG.BUFF = 2) AND NOT "RECIRCULATION DB".MFG.PAUSE));
END_REGION

REGION Network 51: PBV-79 BASKET FILTER INLET
   RUNG wire#powerrail
      Contact( "AlwaysTRUE" )
      { S7_Templates := "SrcType := Int" } NE_Contact(in1 := "MODE SELECTION DB"."MODE BUFF", in2 := 0)
      wire#w1
      Contact( "TRANSFER DB".BIT."SUGAR TO PREMIXING"."PBV-79 BASKET FILTER INLET" )
      wire#w2
      Coil( "TRANSFER DB".OUTPUT."PBV-79 BASKET FILTER INLET" )
   END_RUNG
   RUNG wire#w1
      Contact( "TRANSFER DB".BIT."SUGAR TO MFG"."PBV-79 BASKET FILTER INLET" )
   END_RUNG wire#w2
   // the same network as SCL:
   "TRANSFER DB".OUTPUT."PBV-79 BASKET FILTER INLET" := "AlwaysTRUE" AND ("MODE SELECTION DB"."MODE BUFF" <> 0) AND ("TRANSFER DB".BIT."SUGAR TO PREMIXING"."PBV-79 BASKET FILTER INLET" OR "TRANSFER DB".BIT."SUGAR TO MFG"."PBV-79 BASKET FILTER INLET");
END_REGION

REGION Network 52: PBV-80 BOTTOM OUTLET TO BASKET FILTER
   RUNG wire#powerrail
      Contact( "AlwaysTRUE" )
      { S7_Templates := "SrcType := Int" } NE_Contact(in1 := "MODE SELECTION DB"."MODE BUFF", in2 := 0)
      wire#w1
      Contact( "TRANSFER DB".BIT."SUGAR TO PREMIXING"."PBV-80 BOTTOM OUTLET TO BASKET FILTER" )
      wire#w2
      Coil( "TRANSFER DB".OUTPUT."PBV-80 BOTTOM OUTLET TO BASKET FILTER" )
   END_RUNG
   RUNG wire#w1
      Contact( "TRANSFER DB".BIT."SUGAR TO MFG"."PBV-80 BOTTOM OUTLET TO BASKET FILTER" )
   END_RUNG wire#w2
   // the same network as SCL:
   "TRANSFER DB".OUTPUT."PBV-80 BOTTOM OUTLET TO BASKET FILTER" := "AlwaysTRUE" AND ("MODE SELECTION DB"."MODE BUFF" <> 0) AND ("TRANSFER DB".BIT."SUGAR TO PREMIXING"."PBV-80 BOTTOM OUTLET TO BASKET FILTER" OR "TRANSFER DB".BIT."SUGAR TO MFG"."PBV-80 BOTTOM OUTLET TO BASKET FILTER");
END_REGION

REGION Network 53: PBV-81 TANK BOTTOM OUTLET TO CIP OUTLET
   RUNG wire#powerrail
      Contact( "AlwaysFALSE" )
      { S7_Templates := "SrcType := Int" } NE_Contact(in1 := "MODE SELECTION DB"."MODE BUFF", in2 := 0)
      Coil( "TRANSFER DB".OUTPUT."PBV-81 TANK BOTTOM OUTLET TO CIP OUTLET" )
   END_RUNG
   // the same network as SCL:
   "TRANSFER DB".OUTPUT."PBV-81 TANK BOTTOM OUTLET TO CIP OUTLET" := "AlwaysFALSE" AND ("MODE SELECTION DB"."MODE BUFF" <> 0);
END_REGION

REGION Network 54: PBV-82 CIP ISOLATION
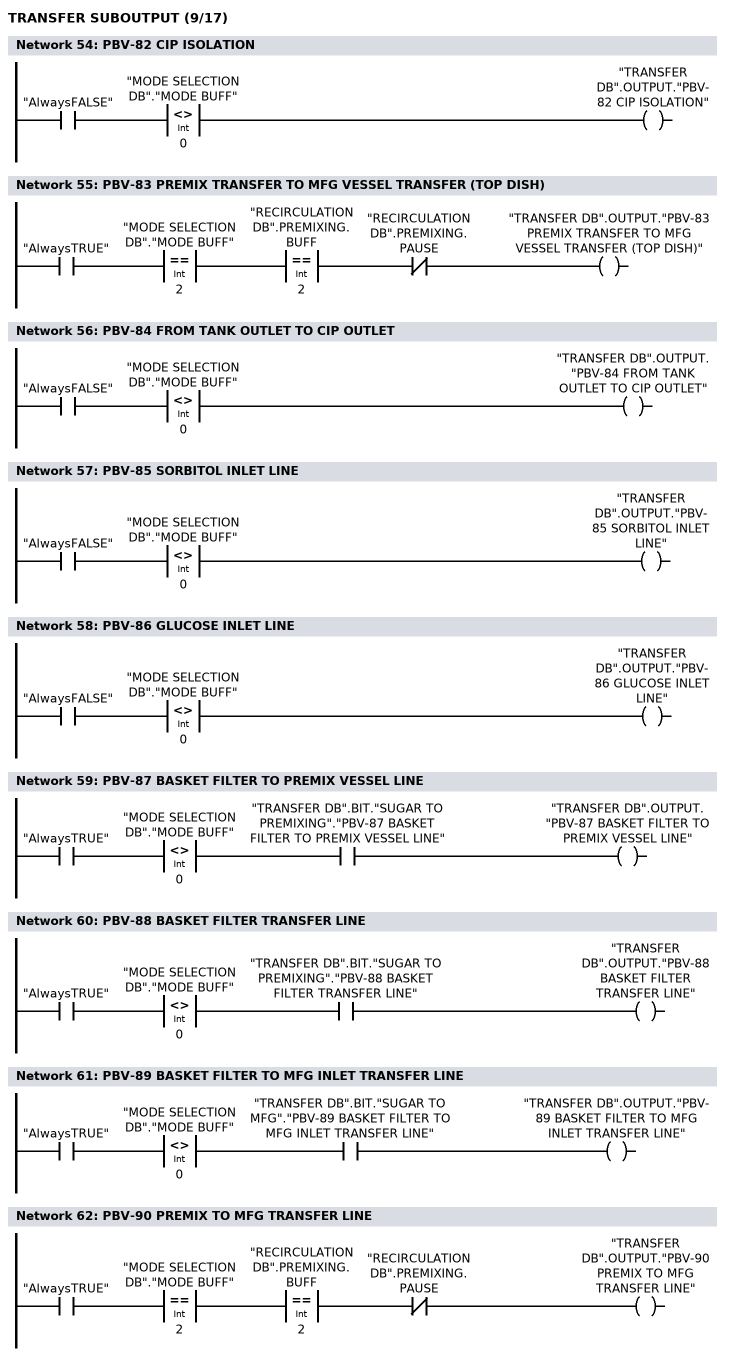
   RUNG wire#powerrail
      Contact( "AlwaysFALSE" )
      { S7_Templates := "SrcType := Int" } NE_Contact(in1 := "MODE SELECTION DB"."MODE BUFF", in2 := 0)
      Coil( "TRANSFER DB".OUTPUT."PBV-82 CIP ISOLATION" )
   END_RUNG
   // the same network as SCL:
   "TRANSFER DB".OUTPUT."PBV-82 CIP ISOLATION" := "AlwaysFALSE" AND ("MODE SELECTION DB"."MODE BUFF" <> 0);
END_REGION

REGION Network 55: PBV-83 PREMIX TRANSFER TO MFG VESSEL TRANSFER (TOP DISH)
   RUNG wire#powerrail
      Contact( "AlwaysTRUE" )
      { S7_Templates := "SrcType := Int" } EQ_Contact(in1 := "MODE SELECTION DB"."MODE BUFF", in2 := 2)
      { S7_Templates := "SrcType := Int" } EQ_Contact(in1 := "RECIRCULATION DB".PREMIXING.BUFF, in2 := 2)
      I_Contact( "RECIRCULATION DB".PREMIXING.PAUSE )
      Coil( "TRANSFER DB".OUTPUT."PBV-83 PREMIX TRANSFER TO MFG VESSEL TRANSFER (TOP DISH)" )
   END_RUNG
   // the same network as SCL:
   "TRANSFER DB".OUTPUT."PBV-83 PREMIX TRANSFER TO MFG VESSEL TRANSFER (TOP DISH)" := "AlwaysTRUE" AND ("MODE SELECTION DB"."MODE BUFF" = 2) AND ("RECIRCULATION DB".PREMIXING.BUFF = 2) AND NOT "RECIRCULATION DB".PREMIXING.PAUSE;
END_REGION

REGION Network 56: PBV-84 FROM TANK OUTLET TO CIP OUTLET
   RUNG wire#powerrail
      Contact( "AlwaysFALSE" )
      { S7_Templates := "SrcType := Int" } NE_Contact(in1 := "MODE SELECTION DB"."MODE BUFF", in2 := 0)
      Coil( "TRANSFER DB".OUTPUT."PBV-84 FROM TANK OUTLET TO CIP OUTLET" )
   END_RUNG
   // the same network as SCL:
   "TRANSFER DB".OUTPUT."PBV-84 FROM TANK OUTLET TO CIP OUTLET" := "AlwaysFALSE" AND ("MODE SELECTION DB"."MODE BUFF" <> 0);
END_REGION

REGION Network 57: PBV-85 SORBITOL INLET LINE
   RUNG wire#powerrail
      Contact( "AlwaysFALSE" )
      { S7_Templates := "SrcType := Int" } NE_Contact(in1 := "MODE SELECTION DB"."MODE BUFF", in2 := 0)
      Coil( "TRANSFER DB".OUTPUT."PBV-85 SORBITOL INLET LINE" )
   END_RUNG
   // the same network as SCL:
   "TRANSFER DB".OUTPUT."PBV-85 SORBITOL INLET LINE" := "AlwaysFALSE" AND ("MODE SELECTION DB"."MODE BUFF" <> 0);
END_REGION

REGION Network 58: PBV-86 GLUCOSE INLET LINE
   RUNG wire#powerrail
      Contact( "AlwaysFALSE" )
      { S7_Templates := "SrcType := Int" } NE_Contact(in1 := "MODE SELECTION DB"."MODE BUFF", in2 := 0)
      Coil( "TRANSFER DB".OUTPUT."PBV-86 GLUCOSE INLET LINE" )
   END_RUNG
   // the same network as SCL:
   "TRANSFER DB".OUTPUT."PBV-86 GLUCOSE INLET LINE" := "AlwaysFALSE" AND ("MODE SELECTION DB"."MODE BUFF" <> 0);
END_REGION

REGION Network 59: PBV-87 BASKET FILTER TO PREMIX VESSEL LINE
   RUNG wire#powerrail
      Contact( "AlwaysTRUE" )
      { S7_Templates := "SrcType := Int" } NE_Contact(in1 := "MODE SELECTION DB"."MODE BUFF", in2 := 0)
      Contact( "TRANSFER DB".BIT."SUGAR TO PREMIXING"."PBV-87 BASKET FILTER TO PREMIX VESSEL LINE" )
      Coil( "TRANSFER DB".OUTPUT."PBV-87 BASKET FILTER TO PREMIX VESSEL LINE" )
   END_RUNG
   // the same network as SCL:
   "TRANSFER DB".OUTPUT."PBV-87 BASKET FILTER TO PREMIX VESSEL LINE" := "AlwaysTRUE" AND ("MODE SELECTION DB"."MODE BUFF" <> 0) AND "TRANSFER DB".BIT."SUGAR TO PREMIXING"."PBV-87 BASKET FILTER TO PREMIX VESSEL LINE";
END_REGION

REGION Network 60: PBV-88 BASKET FILTER TRANSFER LINE
   RUNG wire#powerrail
      Contact( "AlwaysTRUE" )
      { S7_Templates := "SrcType := Int" } NE_Contact(in1 := "MODE SELECTION DB"."MODE BUFF", in2 := 0)
      Contact( "TRANSFER DB".BIT."SUGAR TO PREMIXING"."PBV-88 BASKET FILTER TRANSFER LINE" )
      Coil( "TRANSFER DB".OUTPUT."PBV-88 BASKET FILTER TRANSFER LINE" )
   END_RUNG
   // the same network as SCL:
   "TRANSFER DB".OUTPUT."PBV-88 BASKET FILTER TRANSFER LINE" := "AlwaysTRUE" AND ("MODE SELECTION DB"."MODE BUFF" <> 0) AND "TRANSFER DB".BIT."SUGAR TO PREMIXING"."PBV-88 BASKET FILTER TRANSFER LINE";
END_REGION

REGION Network 61: PBV-89 BASKET FILTER TO MFG INLET TRANSFER LINE
   RUNG wire#powerrail
      Contact( "AlwaysTRUE" )
      { S7_Templates := "SrcType := Int" } NE_Contact(in1 := "MODE SELECTION DB"."MODE BUFF", in2 := 0)
      Contact( "TRANSFER DB".BIT."SUGAR TO MFG"."PBV-89 BASKET FILTER TO MFG INLET TRANSFER LINE" )
      Coil( "TRANSFER DB".OUTPUT."PBV-89 BASKET FILTER TO MFG INLET TRANSFER LINE" )
   END_RUNG
   // the same network as SCL:
   "TRANSFER DB".OUTPUT."PBV-89 BASKET FILTER TO MFG INLET TRANSFER LINE" := "AlwaysTRUE" AND ("MODE SELECTION DB"."MODE BUFF" <> 0) AND "TRANSFER DB".BIT."SUGAR TO MFG"."PBV-89 BASKET FILTER TO MFG INLET TRANSFER LINE";
END_REGION

REGION Network 62: PBV-90 PREMIX TO MFG TRANSFER LINE
   RUNG wire#powerrail
      Contact( "AlwaysTRUE" )
      { S7_Templates := "SrcType := Int" } EQ_Contact(in1 := "MODE SELECTION DB"."MODE BUFF", in2 := 2)
      { S7_Templates := "SrcType := Int" } EQ_Contact(in1 := "RECIRCULATION DB".PREMIXING.BUFF, in2 := 2)
      I_Contact( "RECIRCULATION DB".PREMIXING.PAUSE )
      Coil( "TRANSFER DB".OUTPUT."PBV-90 PREMIX TO MFG TRANSFER LINE" )
   END_RUNG
   // the same network as SCL:
   "TRANSFER DB".OUTPUT."PBV-90 PREMIX TO MFG TRANSFER LINE" := "AlwaysTRUE" AND ("MODE SELECTION DB"."MODE BUFF" = 2) AND ("RECIRCULATION DB".PREMIXING.BUFF = 2) AND NOT "RECIRCULATION DB".PREMIXING.PAUSE;
END_REGION

REGION Network 63: PBV-91 PREMIX TO MFG TRANSFER LINE
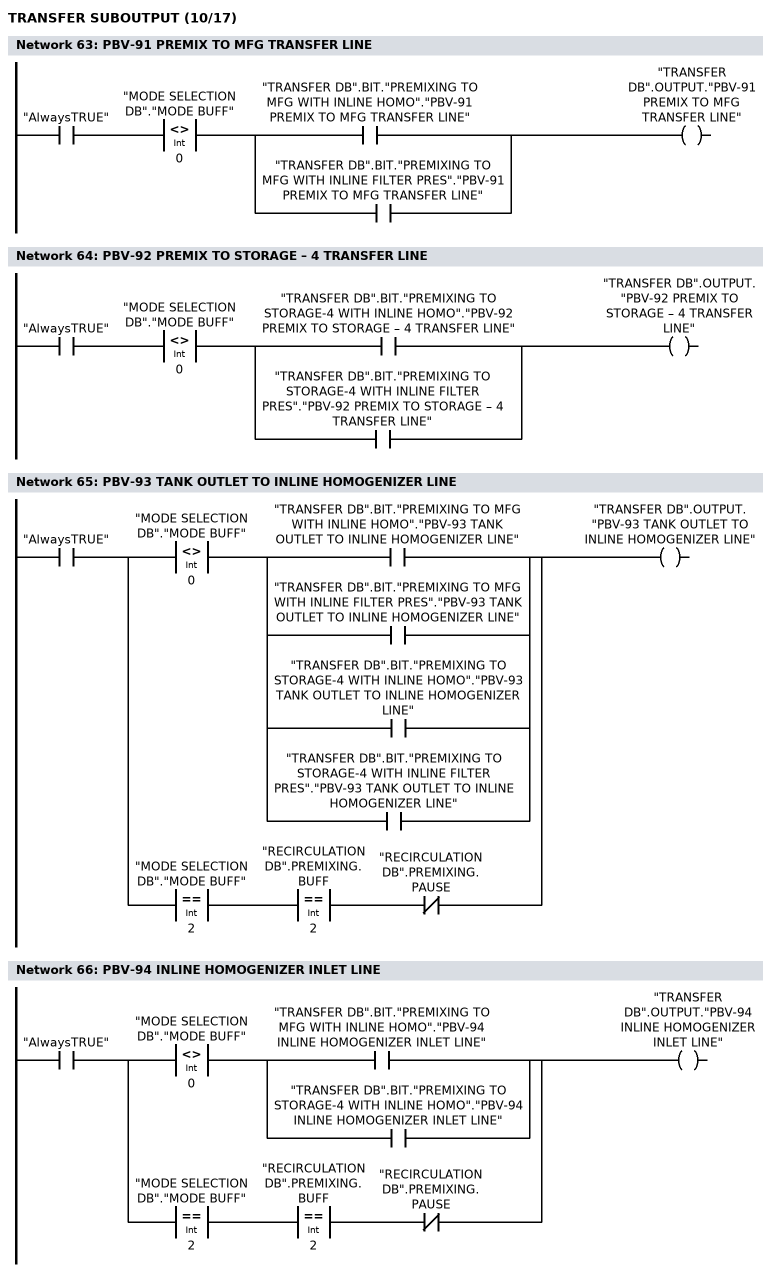
   RUNG wire#powerrail
      Contact( "AlwaysTRUE" )
      { S7_Templates := "SrcType := Int" } NE_Contact(in1 := "MODE SELECTION DB"."MODE BUFF", in2 := 0)
      wire#w1
      Contact( "TRANSFER DB".BIT."PREMIXING TO MFG WITH INLINE HOMO"."PBV-91 PREMIX TO MFG TRANSFER LINE" )
      wire#w2
      Coil( "TRANSFER DB".OUTPUT."PBV-91 PREMIX TO MFG TRANSFER LINE" )
   END_RUNG
   RUNG wire#w1
      Contact( "TRANSFER DB".BIT."PREMIXING TO MFG WITH INLINE FILTER PRES"."PBV-91 PREMIX TO MFG TRANSFER LINE" )
   END_RUNG wire#w2
   // the same network as SCL:
   "TRANSFER DB".OUTPUT."PBV-91 PREMIX TO MFG TRANSFER LINE" := "AlwaysTRUE" AND ("MODE SELECTION DB"."MODE BUFF" <> 0) AND ("TRANSFER DB".BIT."PREMIXING TO MFG WITH INLINE HOMO"."PBV-91 PREMIX TO MFG TRANSFER LINE" OR "TRANSFER DB".BIT."PREMIXING TO MFG WITH INLINE FILTER PRES"."PBV-91 PREMIX TO MFG TRANSFER LINE");
END_REGION

REGION Network 64: PBV-92 PREMIX TO STORAGE – 4 TRANSFER LINE
   RUNG wire#powerrail
      Contact( "AlwaysTRUE" )
      { S7_Templates := "SrcType := Int" } NE_Contact(in1 := "MODE SELECTION DB"."MODE BUFF", in2 := 0)
      wire#w1
      Contact( "TRANSFER DB".BIT."PREMIXING TO STORAGE-4 WITH INLINE HOMO"."PBV-92 PREMIX TO STORAGE – 4 TRANSFER LINE" )
      wire#w2
      Coil( "TRANSFER DB".OUTPUT."PBV-92 PREMIX TO STORAGE – 4 TRANSFER LINE" )
   END_RUNG
   RUNG wire#w1
      Contact( "TRANSFER DB".BIT."PREMIXING TO STORAGE-4 WITH INLINE FILTER PRES"."PBV-92 PREMIX TO STORAGE – 4 TRANSFER LINE" )
   END_RUNG wire#w2
   // the same network as SCL:
   "TRANSFER DB".OUTPUT."PBV-92 PREMIX TO STORAGE – 4 TRANSFER LINE" := "AlwaysTRUE" AND ("MODE SELECTION DB"."MODE BUFF" <> 0) AND ("TRANSFER DB".BIT."PREMIXING TO STORAGE-4 WITH INLINE HOMO"."PBV-92 PREMIX TO STORAGE – 4 TRANSFER LINE" OR "TRANSFER DB".BIT."PREMIXING TO STORAGE-4 WITH INLINE FILTER PRES"."PBV-92 PREMIX TO STORAGE – 4 TRANSFER LINE");
END_REGION

REGION Network 65: PBV-93 TANK OUTLET TO INLINE HOMOGENIZER LINE
   RUNG wire#powerrail
      Contact( "AlwaysTRUE" )
      wire#w1
      { S7_Templates := "SrcType := Int" } NE_Contact(in1 := "MODE SELECTION DB"."MODE BUFF", in2 := 0)
      wire#w2
      Contact( "TRANSFER DB".BIT."PREMIXING TO MFG WITH INLINE HOMO"."PBV-93 TANK OUTLET TO INLINE HOMOGENIZER LINE" )
      wire#w3
      Coil( "TRANSFER DB".OUTPUT."PBV-93 TANK OUTLET TO INLINE HOMOGENIZER LINE" )
   END_RUNG
   RUNG wire#w2
      Contact( "TRANSFER DB".BIT."PREMIXING TO MFG WITH INLINE FILTER PRES"."PBV-93 TANK OUTLET TO INLINE HOMOGENIZER LINE" )
   END_RUNG wire#w3
   RUNG wire#w2
      Contact( "TRANSFER DB".BIT."PREMIXING TO STORAGE-4 WITH INLINE HOMO"."PBV-93 TANK OUTLET TO INLINE HOMOGENIZER LINE" )
   END_RUNG wire#w3
   RUNG wire#w2
      Contact( "TRANSFER DB".BIT."PREMIXING TO STORAGE-4 WITH INLINE FILTER PRES"."PBV-93 TANK OUTLET TO INLINE HOMOGENIZER LINE" )
   END_RUNG wire#w3
   RUNG wire#w1
      { S7_Templates := "SrcType := Int" } EQ_Contact(in1 := "MODE SELECTION DB"."MODE BUFF", in2 := 2)
      { S7_Templates := "SrcType := Int" } EQ_Contact(in1 := "RECIRCULATION DB".PREMIXING.BUFF, in2 := 2)
      I_Contact( "RECIRCULATION DB".PREMIXING.PAUSE )
   END_RUNG wire#w3
   // the same network as SCL:
   "TRANSFER DB".OUTPUT."PBV-93 TANK OUTLET TO INLINE HOMOGENIZER LINE" := "AlwaysTRUE" AND ((("MODE SELECTION DB"."MODE BUFF" <> 0) AND ("TRANSFER DB".BIT."PREMIXING TO MFG WITH INLINE HOMO"."PBV-93 TANK OUTLET TO INLINE HOMOGENIZER LINE" OR "TRANSFER DB".BIT."PREMIXING TO MFG WITH INLINE FILTER PRES"."PBV-93 TANK OUTLET TO INLINE HOMOGENIZER LINE" OR "TRANSFER DB".BIT."PREMIXING TO STORAGE-4 WITH INLINE HOMO"."PBV-93 TANK OUTLET TO INLINE HOMOGENIZER LINE" OR "TRANSFER DB".BIT."PREMIXING TO STORAGE-4 WITH INLINE FILTER PRES"."PBV-93 TANK OUTLET TO INLINE HOMOGENIZER LINE")) OR (("MODE SELECTION DB"."MODE BUFF" = 2) AND ("RECIRCULATION DB".PREMIXING.BUFF = 2) AND NOT "RECIRCULATION DB".PREMIXING.PAUSE));
END_REGION

REGION Network 66: PBV-94 INLINE HOMOGENIZER INLET LINE
   RUNG wire#powerrail
      Contact( "AlwaysTRUE" )
      wire#w1
      { S7_Templates := "SrcType := Int" } NE_Contact(in1 := "MODE SELECTION DB"."MODE BUFF", in2 := 0)
      wire#w2
      Contact( "TRANSFER DB".BIT."PREMIXING TO MFG WITH INLINE HOMO"."PBV-94 INLINE HOMOGENIZER INLET LINE" )
      wire#w3
      Coil( "TRANSFER DB".OUTPUT."PBV-94 INLINE HOMOGENIZER INLET LINE" )
   END_RUNG
   RUNG wire#w2
      Contact( "TRANSFER DB".BIT."PREMIXING TO STORAGE-4 WITH INLINE HOMO"."PBV-94 INLINE HOMOGENIZER INLET LINE" )
   END_RUNG wire#w3
   RUNG wire#w1
      { S7_Templates := "SrcType := Int" } EQ_Contact(in1 := "MODE SELECTION DB"."MODE BUFF", in2 := 2)
      { S7_Templates := "SrcType := Int" } EQ_Contact(in1 := "RECIRCULATION DB".PREMIXING.BUFF, in2 := 2)
      I_Contact( "RECIRCULATION DB".PREMIXING.PAUSE )
   END_RUNG wire#w3
   // the same network as SCL:
   "TRANSFER DB".OUTPUT."PBV-94 INLINE HOMOGENIZER INLET LINE" := "AlwaysTRUE" AND ((("MODE SELECTION DB"."MODE BUFF" <> 0) AND ("TRANSFER DB".BIT."PREMIXING TO MFG WITH INLINE HOMO"."PBV-94 INLINE HOMOGENIZER INLET LINE" OR "TRANSFER DB".BIT."PREMIXING TO STORAGE-4 WITH INLINE HOMO"."PBV-94 INLINE HOMOGENIZER INLET LINE")) OR (("MODE SELECTION DB"."MODE BUFF" = 2) AND ("RECIRCULATION DB".PREMIXING.BUFF = 2) AND NOT "RECIRCULATION DB".PREMIXING.PAUSE));
END_REGION

REGION Network 67: PBV-95 TANK OUTLET TO FILTER PRESS LINE
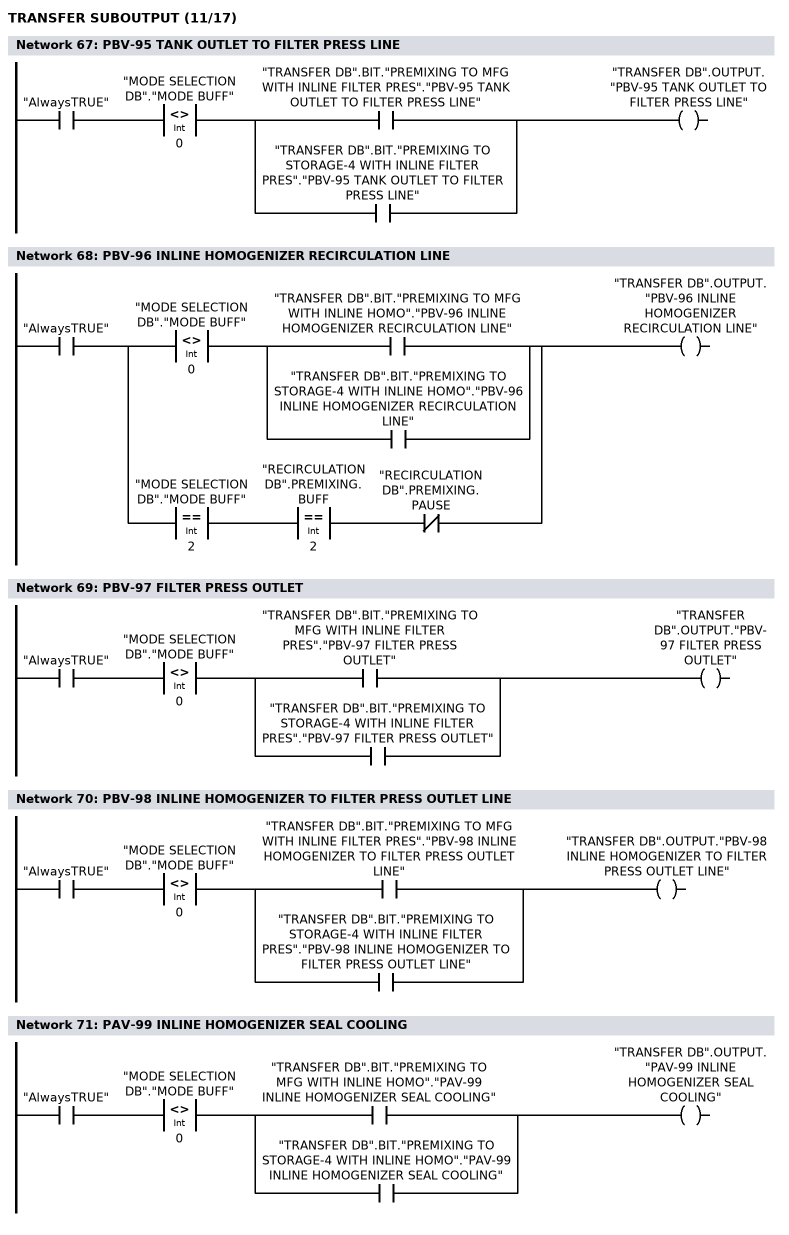
   RUNG wire#powerrail
      Contact( "AlwaysTRUE" )
      { S7_Templates := "SrcType := Int" } NE_Contact(in1 := "MODE SELECTION DB"."MODE BUFF", in2 := 0)
      wire#w1
      Contact( "TRANSFER DB".BIT."PREMIXING TO MFG WITH INLINE FILTER PRES"."PBV-95 TANK OUTLET TO FILTER PRESS LINE" )
      wire#w2
      Coil( "TRANSFER DB".OUTPUT."PBV-95 TANK OUTLET TO FILTER PRESS LINE" )
   END_RUNG
   RUNG wire#w1
      Contact( "TRANSFER DB".BIT."PREMIXING TO STORAGE-4 WITH INLINE FILTER PRES"."PBV-95 TANK OUTLET TO FILTER PRESS LINE" )
   END_RUNG wire#w2
   // the same network as SCL:
   "TRANSFER DB".OUTPUT."PBV-95 TANK OUTLET TO FILTER PRESS LINE" := "AlwaysTRUE" AND ("MODE SELECTION DB"."MODE BUFF" <> 0) AND ("TRANSFER DB".BIT."PREMIXING TO MFG WITH INLINE FILTER PRES"."PBV-95 TANK OUTLET TO FILTER PRESS LINE" OR "TRANSFER DB".BIT."PREMIXING TO STORAGE-4 WITH INLINE FILTER PRES"."PBV-95 TANK OUTLET TO FILTER PRESS LINE");
END_REGION

REGION Network 68: PBV-96 INLINE HOMOGENIZER RECIRCULATION LINE
   RUNG wire#powerrail
      Contact( "AlwaysTRUE" )
      wire#w1
      { S7_Templates := "SrcType := Int" } NE_Contact(in1 := "MODE SELECTION DB"."MODE BUFF", in2 := 0)
      wire#w2
      Contact( "TRANSFER DB".BIT."PREMIXING TO MFG WITH INLINE HOMO"."PBV-96 INLINE HOMOGENIZER RECIRCULATION LINE" )
      wire#w3
      Coil( "TRANSFER DB".OUTPUT."PBV-96 INLINE HOMOGENIZER RECIRCULATION LINE" )
   END_RUNG
   RUNG wire#w2
      Contact( "TRANSFER DB".BIT."PREMIXING TO STORAGE-4 WITH INLINE HOMO"."PBV-96 INLINE HOMOGENIZER RECIRCULATION LINE" )
   END_RUNG wire#w3
   RUNG wire#w1
      { S7_Templates := "SrcType := Int" } EQ_Contact(in1 := "MODE SELECTION DB"."MODE BUFF", in2 := 2)
      { S7_Templates := "SrcType := Int" } EQ_Contact(in1 := "RECIRCULATION DB".PREMIXING.BUFF, in2 := 2)
      I_Contact( "RECIRCULATION DB".PREMIXING.PAUSE )
   END_RUNG wire#w3
   // the same network as SCL:
   "TRANSFER DB".OUTPUT."PBV-96 INLINE HOMOGENIZER RECIRCULATION LINE" := "AlwaysTRUE" AND ((("MODE SELECTION DB"."MODE BUFF" <> 0) AND ("TRANSFER DB".BIT."PREMIXING TO MFG WITH INLINE HOMO"."PBV-96 INLINE HOMOGENIZER RECIRCULATION LINE" OR "TRANSFER DB".BIT."PREMIXING TO STORAGE-4 WITH INLINE HOMO"."PBV-96 INLINE HOMOGENIZER RECIRCULATION LINE")) OR (("MODE SELECTION DB"."MODE BUFF" = 2) AND ("RECIRCULATION DB".PREMIXING.BUFF = 2) AND NOT "RECIRCULATION DB".PREMIXING.PAUSE));
END_REGION

REGION Network 69: PBV-97 FILTER PRESS OUTLET
   RUNG wire#powerrail
      Contact( "AlwaysTRUE" )
      { S7_Templates := "SrcType := Int" } NE_Contact(in1 := "MODE SELECTION DB"."MODE BUFF", in2 := 0)
      wire#w1
      Contact( "TRANSFER DB".BIT."PREMIXING TO MFG WITH INLINE FILTER PRES"."PBV-97 FILTER PRESS OUTLET" )
      wire#w2
      Coil( "TRANSFER DB".OUTPUT."PBV-97 FILTER PRESS OUTLET" )
   END_RUNG
   RUNG wire#w1
      Contact( "TRANSFER DB".BIT."PREMIXING TO STORAGE-4 WITH INLINE FILTER PRES"."PBV-97 FILTER PRESS OUTLET" )
   END_RUNG wire#w2
   // the same network as SCL:
   "TRANSFER DB".OUTPUT."PBV-97 FILTER PRESS OUTLET" := "AlwaysTRUE" AND ("MODE SELECTION DB"."MODE BUFF" <> 0) AND ("TRANSFER DB".BIT."PREMIXING TO MFG WITH INLINE FILTER PRES"."PBV-97 FILTER PRESS OUTLET" OR "TRANSFER DB".BIT."PREMIXING TO STORAGE-4 WITH INLINE FILTER PRES"."PBV-97 FILTER PRESS OUTLET");
END_REGION

REGION Network 70: PBV-98 INLINE HOMOGENIZER TO FILTER PRESS OUTLET LINE
   RUNG wire#powerrail
      Contact( "AlwaysTRUE" )
      { S7_Templates := "SrcType := Int" } NE_Contact(in1 := "MODE SELECTION DB"."MODE BUFF", in2 := 0)
      wire#w1
      Contact( "TRANSFER DB".BIT."PREMIXING TO MFG WITH INLINE FILTER PRES"."PBV-98 INLINE HOMOGENIZER TO FILTER PRESS OUTLET LINE" )
      wire#w2
      Coil( "TRANSFER DB".OUTPUT."PBV-98 INLINE HOMOGENIZER TO FILTER PRESS OUTLET LINE" )
   END_RUNG
   RUNG wire#w1
      Contact( "TRANSFER DB".BIT."PREMIXING TO STORAGE-4 WITH INLINE FILTER PRES"."PBV-98 INLINE HOMOGENIZER TO FILTER PRESS OUTLET LINE" )
   END_RUNG wire#w2
   // the same network as SCL:
   "TRANSFER DB".OUTPUT."PBV-98 INLINE HOMOGENIZER TO FILTER PRESS OUTLET LINE" := "AlwaysTRUE" AND ("MODE SELECTION DB"."MODE BUFF" <> 0) AND ("TRANSFER DB".BIT."PREMIXING TO MFG WITH INLINE FILTER PRES"."PBV-98 INLINE HOMOGENIZER TO FILTER PRESS OUTLET LINE" OR "TRANSFER DB".BIT."PREMIXING TO STORAGE-4 WITH INLINE FILTER PRES"."PBV-98 INLINE HOMOGENIZER TO FILTER PRESS OUTLET LINE");
END_REGION

REGION Network 71: PAV-99 INLINE HOMOGENIZER SEAL COOLING
   RUNG wire#powerrail
      Contact( "AlwaysTRUE" )
      { S7_Templates := "SrcType := Int" } NE_Contact(in1 := "MODE SELECTION DB"."MODE BUFF", in2 := 0)
      wire#w1
      Contact( "TRANSFER DB".BIT."PREMIXING TO MFG WITH INLINE HOMO"."PAV-99 INLINE HOMOGENIZER SEAL COOLING" )
      wire#w2
      Coil( "TRANSFER DB".OUTPUT."PAV-99 INLINE HOMOGENIZER SEAL COOLING" )
   END_RUNG
   RUNG wire#w1
      Contact( "TRANSFER DB".BIT."PREMIXING TO STORAGE-4 WITH INLINE HOMO"."PAV-99 INLINE HOMOGENIZER SEAL COOLING" )
   END_RUNG wire#w2
   // the same network as SCL:
   "TRANSFER DB".OUTPUT."PAV-99 INLINE HOMOGENIZER SEAL COOLING" := "AlwaysTRUE" AND ("MODE SELECTION DB"."MODE BUFF" <> 0) AND ("TRANSFER DB".BIT."PREMIXING TO MFG WITH INLINE HOMO"."PAV-99 INLINE HOMOGENIZER SEAL COOLING" OR "TRANSFER DB".BIT."PREMIXING TO STORAGE-4 WITH INLINE HOMO"."PAV-99 INLINE HOMOGENIZER SEAL COOLING");
END_REGION

REGION Network 72: PBV-100 FILTER PRESS INLET
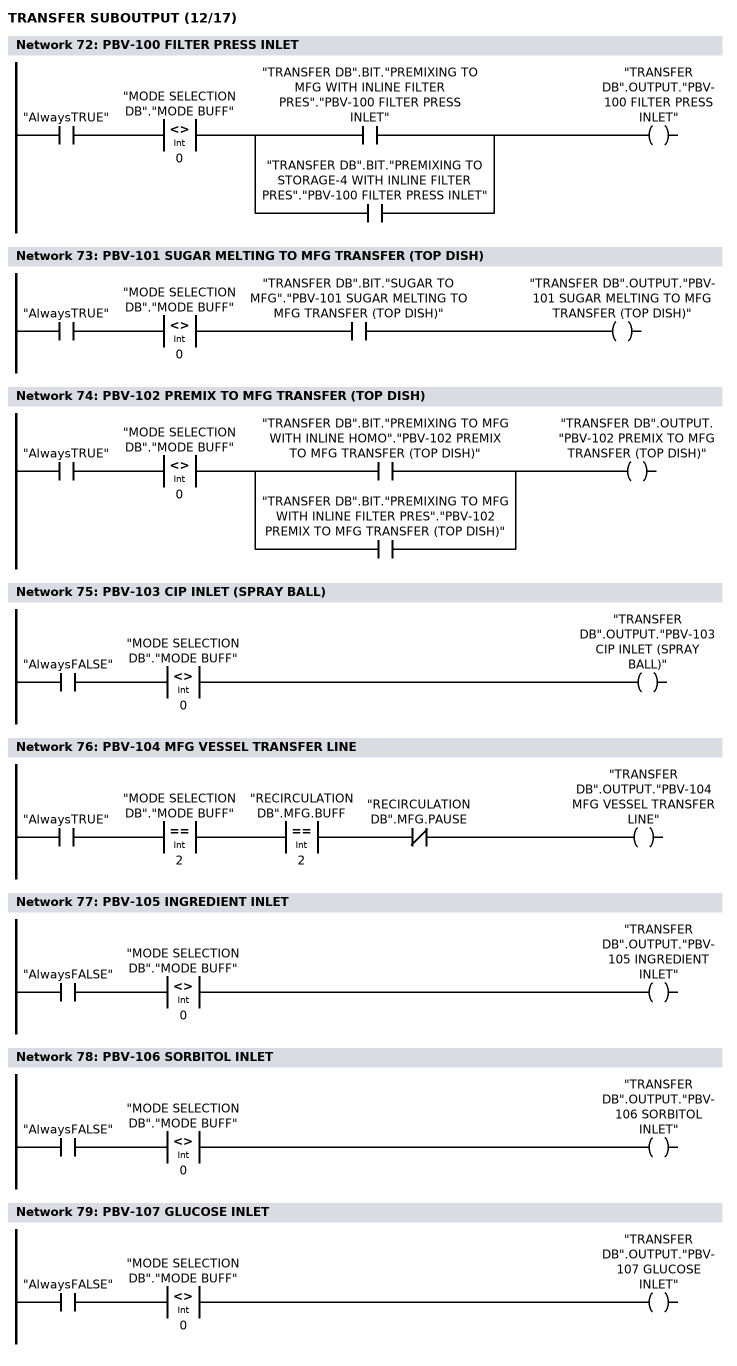
   RUNG wire#powerrail
      Contact( "AlwaysTRUE" )
      { S7_Templates := "SrcType := Int" } NE_Contact(in1 := "MODE SELECTION DB"."MODE BUFF", in2 := 0)
      wire#w1
      Contact( "TRANSFER DB".BIT."PREMIXING TO MFG WITH INLINE FILTER PRES"."PBV-100 FILTER PRESS INLET" )
      wire#w2
      Coil( "TRANSFER DB".OUTPUT."PBV-100 FILTER PRESS INLET" )
   END_RUNG
   RUNG wire#w1
      Contact( "TRANSFER DB".BIT."PREMIXING TO STORAGE-4 WITH INLINE FILTER PRES"."PBV-100 FILTER PRESS INLET" )
   END_RUNG wire#w2
   // the same network as SCL:
   "TRANSFER DB".OUTPUT."PBV-100 FILTER PRESS INLET" := "AlwaysTRUE" AND ("MODE SELECTION DB"."MODE BUFF" <> 0) AND ("TRANSFER DB".BIT."PREMIXING TO MFG WITH INLINE FILTER PRES"."PBV-100 FILTER PRESS INLET" OR "TRANSFER DB".BIT."PREMIXING TO STORAGE-4 WITH INLINE FILTER PRES"."PBV-100 FILTER PRESS INLET");
END_REGION

REGION Network 73: PBV-101 SUGAR MELTING TO MFG TRANSFER (TOP DISH)
   RUNG wire#powerrail
      Contact( "AlwaysTRUE" )
      { S7_Templates := "SrcType := Int" } NE_Contact(in1 := "MODE SELECTION DB"."MODE BUFF", in2 := 0)
      Contact( "TRANSFER DB".BIT."SUGAR TO MFG"."PBV-101 SUGAR MELTING TO MFG TRANSFER (TOP DISH)" )
      Coil( "TRANSFER DB".OUTPUT."PBV-101 SUGAR MELTING TO MFG TRANSFER (TOP DISH)" )
   END_RUNG
   // the same network as SCL:
   "TRANSFER DB".OUTPUT."PBV-101 SUGAR MELTING TO MFG TRANSFER (TOP DISH)" := "AlwaysTRUE" AND ("MODE SELECTION DB"."MODE BUFF" <> 0) AND "TRANSFER DB".BIT."SUGAR TO MFG"."PBV-101 SUGAR MELTING TO MFG TRANSFER (TOP DISH)";
END_REGION

REGION Network 74: PBV-102 PREMIX TO MFG TRANSFER (TOP DISH)
   RUNG wire#powerrail
      Contact( "AlwaysTRUE" )
      { S7_Templates := "SrcType := Int" } NE_Contact(in1 := "MODE SELECTION DB"."MODE BUFF", in2 := 0)
      wire#w1
      Contact( "TRANSFER DB".BIT."PREMIXING TO MFG WITH INLINE HOMO"."PBV-102 PREMIX TO MFG TRANSFER (TOP DISH)" )
      wire#w2
      Coil( "TRANSFER DB".OUTPUT."PBV-102 PREMIX TO MFG TRANSFER (TOP DISH)" )
   END_RUNG
   RUNG wire#w1
      Contact( "TRANSFER DB".BIT."PREMIXING TO MFG WITH INLINE FILTER PRES"."PBV-102 PREMIX TO MFG TRANSFER (TOP DISH)" )
   END_RUNG wire#w2
   // the same network as SCL:
   "TRANSFER DB".OUTPUT."PBV-102 PREMIX TO MFG TRANSFER (TOP DISH)" := "AlwaysTRUE" AND ("MODE SELECTION DB"."MODE BUFF" <> 0) AND ("TRANSFER DB".BIT."PREMIXING TO MFG WITH INLINE HOMO"."PBV-102 PREMIX TO MFG TRANSFER (TOP DISH)" OR "TRANSFER DB".BIT."PREMIXING TO MFG WITH INLINE FILTER PRES"."PBV-102 PREMIX TO MFG TRANSFER (TOP DISH)");
END_REGION

REGION Network 75: PBV-103 CIP INLET (SPRAY BALL)
   RUNG wire#powerrail
      Contact( "AlwaysFALSE" )
      { S7_Templates := "SrcType := Int" } NE_Contact(in1 := "MODE SELECTION DB"."MODE BUFF", in2 := 0)
      Coil( "TRANSFER DB".OUTPUT."PBV-103 CIP INLET (SPRAY BALL)" )
   END_RUNG
   // the same network as SCL:
   "TRANSFER DB".OUTPUT."PBV-103 CIP INLET (SPRAY BALL)" := "AlwaysFALSE" AND ("MODE SELECTION DB"."MODE BUFF" <> 0);
END_REGION

REGION Network 76: PBV-104 MFG VESSEL TRANSFER LINE
   RUNG wire#powerrail
      Contact( "AlwaysTRUE" )
      { S7_Templates := "SrcType := Int" } EQ_Contact(in1 := "MODE SELECTION DB"."MODE BUFF", in2 := 2)
      { S7_Templates := "SrcType := Int" } EQ_Contact(in1 := "RECIRCULATION DB".MFG.BUFF, in2 := 2)
      I_Contact( "RECIRCULATION DB".MFG.PAUSE )
      Coil( "TRANSFER DB".OUTPUT."PBV-104 MFG VESSEL TRANSFER LINE" )
   END_RUNG
   // the same network as SCL:
   "TRANSFER DB".OUTPUT."PBV-104 MFG VESSEL TRANSFER LINE" := "AlwaysTRUE" AND ("MODE SELECTION DB"."MODE BUFF" = 2) AND ("RECIRCULATION DB".MFG.BUFF = 2) AND NOT "RECIRCULATION DB".MFG.PAUSE;
END_REGION

REGION Network 77: PBV-105 INGREDIENT INLET
   RUNG wire#powerrail
      Contact( "AlwaysFALSE" )
      { S7_Templates := "SrcType := Int" } NE_Contact(in1 := "MODE SELECTION DB"."MODE BUFF", in2 := 0)
      Coil( "TRANSFER DB".OUTPUT."PBV-105 INGREDIENT INLET" )
   END_RUNG
   // the same network as SCL:
   "TRANSFER DB".OUTPUT."PBV-105 INGREDIENT INLET" := "AlwaysFALSE" AND ("MODE SELECTION DB"."MODE BUFF" <> 0);
END_REGION

REGION Network 78: PBV-106 SORBITOL INLET
   RUNG wire#powerrail
      Contact( "AlwaysFALSE" )
      { S7_Templates := "SrcType := Int" } NE_Contact(in1 := "MODE SELECTION DB"."MODE BUFF", in2 := 0)
      Coil( "TRANSFER DB".OUTPUT."PBV-106 SORBITOL INLET" )
   END_RUNG
   // the same network as SCL:
   "TRANSFER DB".OUTPUT."PBV-106 SORBITOL INLET" := "AlwaysFALSE" AND ("MODE SELECTION DB"."MODE BUFF" <> 0);
END_REGION

REGION Network 79: PBV-107 GLUCOSE INLET
   RUNG wire#powerrail
      Contact( "AlwaysFALSE" )
      { S7_Templates := "SrcType := Int" } NE_Contact(in1 := "MODE SELECTION DB"."MODE BUFF", in2 := 0)
      Coil( "TRANSFER DB".OUTPUT."PBV-107 GLUCOSE INLET" )
   END_RUNG
   // the same network as SCL:
   "TRANSFER DB".OUTPUT."PBV-107 GLUCOSE INLET" := "AlwaysFALSE" AND ("MODE SELECTION DB"."MODE BUFF" <> 0);
END_REGION

REGION Network 80: PBV-108 INLINE HOMOGENIZER TO FILTER PRESS INLET LINE
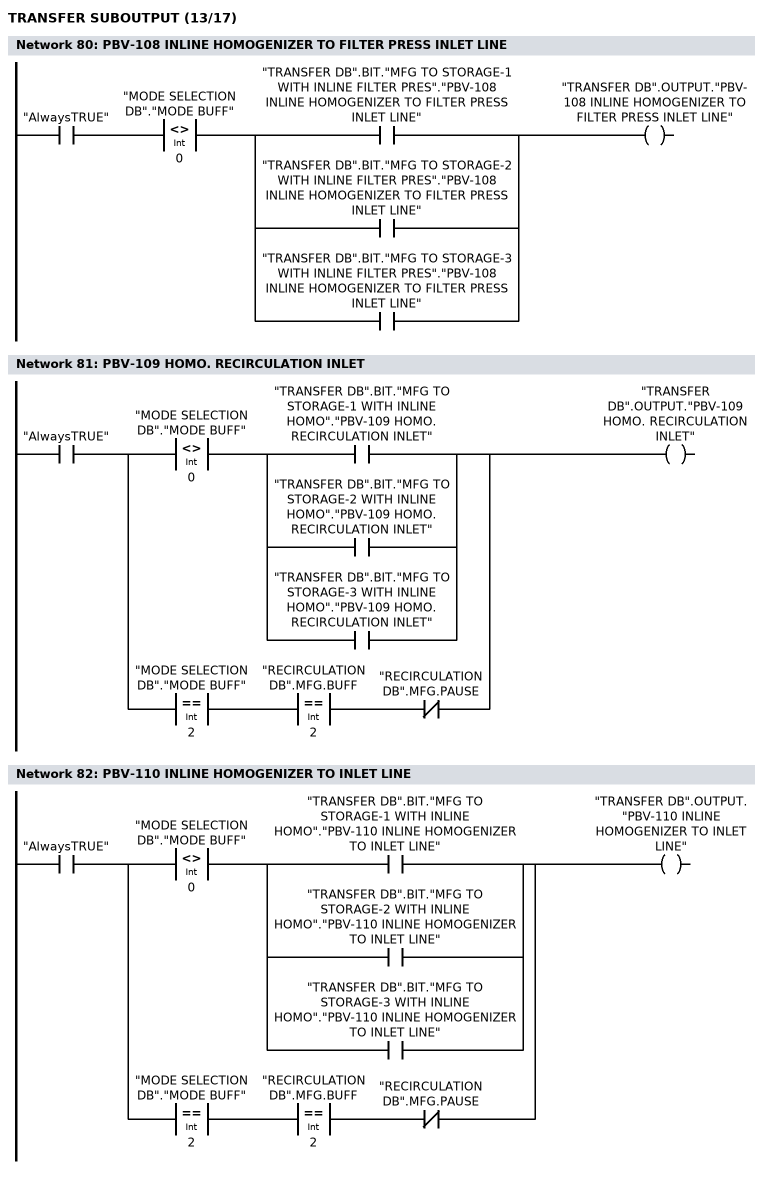
   RUNG wire#powerrail
      Contact( "AlwaysTRUE" )
      { S7_Templates := "SrcType := Int" } NE_Contact(in1 := "MODE SELECTION DB"."MODE BUFF", in2 := 0)
      wire#w1
      Contact( "TRANSFER DB".BIT."MFG TO STORAGE-1 WITH INLINE FILTER PRES"."PBV-108 INLINE HOMOGENIZER TO FILTER PRESS INLET LINE" )
      wire#w2
      Coil( "TRANSFER DB".OUTPUT."PBV-108 INLINE HOMOGENIZER TO FILTER PRESS INLET LINE" )
   END_RUNG
   RUNG wire#w1
      Contact( "TRANSFER DB".BIT."MFG TO STORAGE-2 WITH INLINE FILTER PRES"."PBV-108 INLINE HOMOGENIZER TO FILTER PRESS INLET LINE" )
   END_RUNG wire#w2
   RUNG wire#w1
      Contact( "TRANSFER DB".BIT."MFG TO STORAGE-3 WITH INLINE FILTER PRES"."PBV-108 INLINE HOMOGENIZER TO FILTER PRESS INLET LINE" )
   END_RUNG wire#w2
   // the same network as SCL:
   "TRANSFER DB".OUTPUT."PBV-108 INLINE HOMOGENIZER TO FILTER PRESS INLET LINE" := "AlwaysTRUE" AND ("MODE SELECTION DB"."MODE BUFF" <> 0) AND ("TRANSFER DB".BIT."MFG TO STORAGE-1 WITH INLINE FILTER PRES"."PBV-108 INLINE HOMOGENIZER TO FILTER PRESS INLET LINE" OR "TRANSFER DB".BIT."MFG TO STORAGE-2 WITH INLINE FILTER PRES"."PBV-108 INLINE HOMOGENIZER TO FILTER PRESS INLET LINE" OR "TRANSFER DB".BIT."MFG TO STORAGE-3 WITH INLINE FILTER PRES"."PBV-108 INLINE HOMOGENIZER TO FILTER PRESS INLET LINE");
END_REGION

REGION Network 81: PBV-109 HOMO. RECIRCULATION INLET
   RUNG wire#powerrail
      Contact( "AlwaysTRUE" )
      wire#w1
      { S7_Templates := "SrcType := Int" } NE_Contact(in1 := "MODE SELECTION DB"."MODE BUFF", in2 := 0)
      wire#w2
      Contact( "TRANSFER DB".BIT."MFG TO STORAGE-1 WITH INLINE HOMO"."PBV-109 HOMO. RECIRCULATION INLET" )
      wire#w3
      Coil( "TRANSFER DB".OUTPUT."PBV-109 HOMO. RECIRCULATION INLET" )
   END_RUNG
   RUNG wire#w2
      Contact( "TRANSFER DB".BIT."MFG TO STORAGE-2 WITH INLINE HOMO"."PBV-109 HOMO. RECIRCULATION INLET" )
   END_RUNG wire#w3
   RUNG wire#w2
      Contact( "TRANSFER DB".BIT."MFG TO STORAGE-3 WITH INLINE HOMO"."PBV-109 HOMO. RECIRCULATION INLET" )
   END_RUNG wire#w3
   RUNG wire#w1
      { S7_Templates := "SrcType := Int" } EQ_Contact(in1 := "MODE SELECTION DB"."MODE BUFF", in2 := 2)
      { S7_Templates := "SrcType := Int" } EQ_Contact(in1 := "RECIRCULATION DB".MFG.BUFF, in2 := 2)
      I_Contact( "RECIRCULATION DB".MFG.PAUSE )
   END_RUNG wire#w3
   // the same network as SCL:
   "TRANSFER DB".OUTPUT."PBV-109 HOMO. RECIRCULATION INLET" := "AlwaysTRUE" AND ((("MODE SELECTION DB"."MODE BUFF" <> 0) AND ("TRANSFER DB".BIT."MFG TO STORAGE-1 WITH INLINE HOMO"."PBV-109 HOMO. RECIRCULATION INLET" OR "TRANSFER DB".BIT."MFG TO STORAGE-2 WITH INLINE HOMO"."PBV-109 HOMO. RECIRCULATION INLET" OR "TRANSFER DB".BIT."MFG TO STORAGE-3 WITH INLINE HOMO"."PBV-109 HOMO. RECIRCULATION INLET")) OR (("MODE SELECTION DB"."MODE BUFF" = 2) AND ("RECIRCULATION DB".MFG.BUFF = 2) AND NOT "RECIRCULATION DB".MFG.PAUSE));
END_REGION

REGION Network 82: PBV-110 INLINE HOMOGENIZER TO INLET LINE
   RUNG wire#powerrail
      Contact( "AlwaysTRUE" )
      wire#w1
      { S7_Templates := "SrcType := Int" } NE_Contact(in1 := "MODE SELECTION DB"."MODE BUFF", in2 := 0)
      wire#w2
      Contact( "TRANSFER DB".BIT."MFG TO STORAGE-1 WITH INLINE HOMO"."PBV-110 INLINE HOMOGENIZER TO INLET LINE" )
      wire#w3
      Coil( "TRANSFER DB".OUTPUT."PBV-110 INLINE HOMOGENIZER TO INLET LINE" )
   END_RUNG
   RUNG wire#w2
      Contact( "TRANSFER DB".BIT."MFG TO STORAGE-2 WITH INLINE HOMO"."PBV-110 INLINE HOMOGENIZER TO INLET LINE" )
   END_RUNG wire#w3
   RUNG wire#w2
      Contact( "TRANSFER DB".BIT."MFG TO STORAGE-3 WITH INLINE HOMO"."PBV-110 INLINE HOMOGENIZER TO INLET LINE" )
   END_RUNG wire#w3
   RUNG wire#w1
      { S7_Templates := "SrcType := Int" } EQ_Contact(in1 := "MODE SELECTION DB"."MODE BUFF", in2 := 2)
      { S7_Templates := "SrcType := Int" } EQ_Contact(in1 := "RECIRCULATION DB".MFG.BUFF, in2 := 2)
      I_Contact( "RECIRCULATION DB".MFG.PAUSE )
   END_RUNG wire#w3
   // the same network as SCL:
   "TRANSFER DB".OUTPUT."PBV-110 INLINE HOMOGENIZER TO INLET LINE" := "AlwaysTRUE" AND ((("MODE SELECTION DB"."MODE BUFF" <> 0) AND ("TRANSFER DB".BIT."MFG TO STORAGE-1 WITH INLINE HOMO"."PBV-110 INLINE HOMOGENIZER TO INLET LINE" OR "TRANSFER DB".BIT."MFG TO STORAGE-2 WITH INLINE HOMO"."PBV-110 INLINE HOMOGENIZER TO INLET LINE" OR "TRANSFER DB".BIT."MFG TO STORAGE-3 WITH INLINE HOMO"."PBV-110 INLINE HOMOGENIZER TO INLET LINE")) OR (("MODE SELECTION DB"."MODE BUFF" = 2) AND ("RECIRCULATION DB".MFG.BUFF = 2) AND NOT "RECIRCULATION DB".MFG.PAUSE));
END_REGION

REGION Network 83: PBV-111 FILTER PRESS OUTLER VALVE
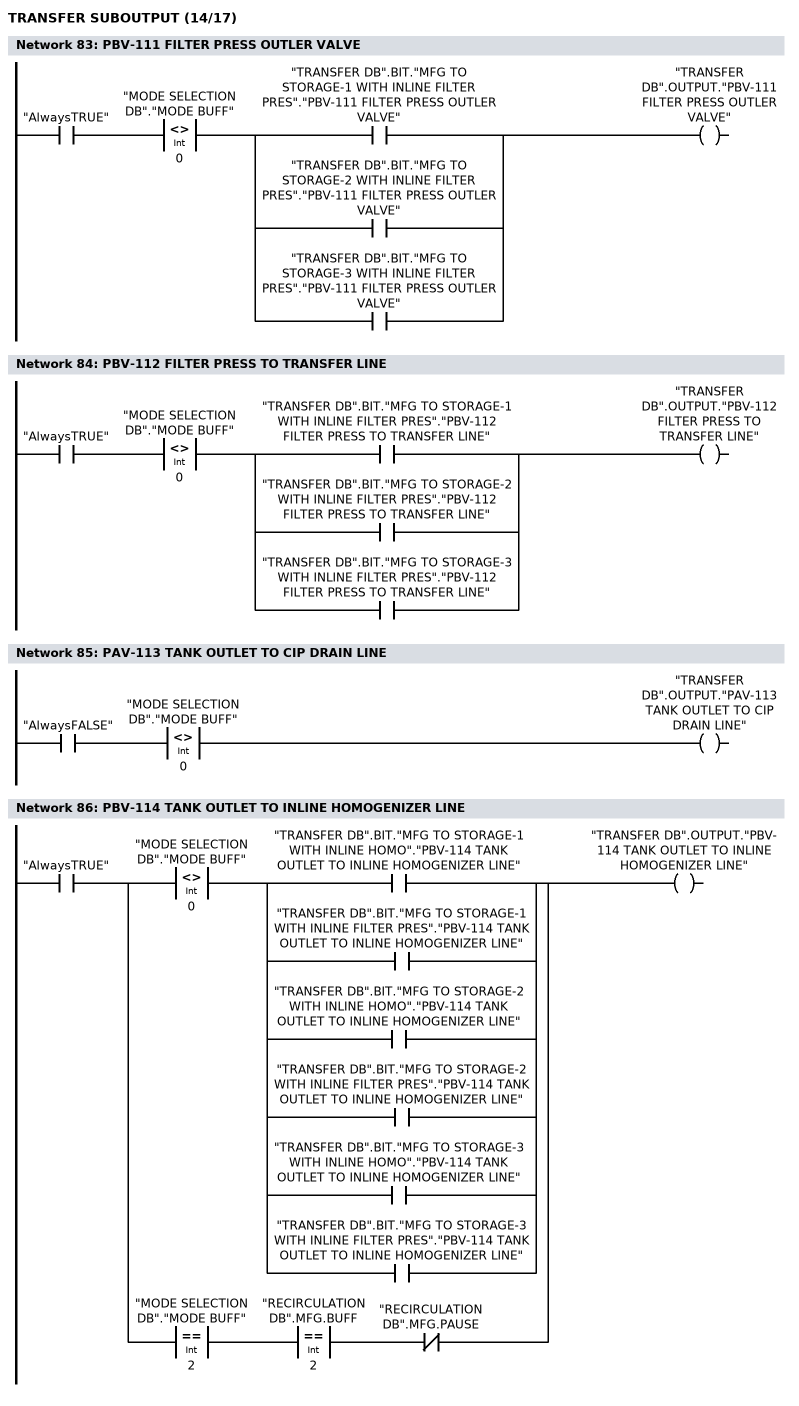
   RUNG wire#powerrail
      Contact( "AlwaysTRUE" )
      { S7_Templates := "SrcType := Int" } NE_Contact(in1 := "MODE SELECTION DB"."MODE BUFF", in2 := 0)
      wire#w1
      Contact( "TRANSFER DB".BIT."MFG TO STORAGE-1 WITH INLINE FILTER PRES"."PBV-111 FILTER PRESS OUTLER VALVE" )
      wire#w2
      Coil( "TRANSFER DB".OUTPUT."PBV-111 FILTER PRESS OUTLER VALVE" )
   END_RUNG
   RUNG wire#w1
      Contact( "TRANSFER DB".BIT."MFG TO STORAGE-2 WITH INLINE FILTER PRES"."PBV-111 FILTER PRESS OUTLER VALVE" )
   END_RUNG wire#w2
   RUNG wire#w1
      Contact( "TRANSFER DB".BIT."MFG TO STORAGE-3 WITH INLINE FILTER PRES"."PBV-111 FILTER PRESS OUTLER VALVE" )
   END_RUNG wire#w2
   // the same network as SCL:
   "TRANSFER DB".OUTPUT."PBV-111 FILTER PRESS OUTLER VALVE" := "AlwaysTRUE" AND ("MODE SELECTION DB"."MODE BUFF" <> 0) AND ("TRANSFER DB".BIT."MFG TO STORAGE-1 WITH INLINE FILTER PRES"."PBV-111 FILTER PRESS OUTLER VALVE" OR "TRANSFER DB".BIT."MFG TO STORAGE-2 WITH INLINE FILTER PRES"."PBV-111 FILTER PRESS OUTLER VALVE" OR "TRANSFER DB".BIT."MFG TO STORAGE-3 WITH INLINE FILTER PRES"."PBV-111 FILTER PRESS OUTLER VALVE");
END_REGION

REGION Network 84: PBV-112 FILTER PRESS TO TRANSFER LINE
   RUNG wire#powerrail
      Contact( "AlwaysTRUE" )
      { S7_Templates := "SrcType := Int" } NE_Contact(in1 := "MODE SELECTION DB"."MODE BUFF", in2 := 0)
      wire#w1
      Contact( "TRANSFER DB".BIT."MFG TO STORAGE-1 WITH INLINE FILTER PRES"."PBV-112 FILTER PRESS TO TRANSFER LINE" )
      wire#w2
      Coil( "TRANSFER DB".OUTPUT."PBV-112 FILTER PRESS TO TRANSFER LINE" )
   END_RUNG
   RUNG wire#w1
      Contact( "TRANSFER DB".BIT."MFG TO STORAGE-2 WITH INLINE FILTER PRES"."PBV-112 FILTER PRESS TO TRANSFER LINE" )
   END_RUNG wire#w2
   RUNG wire#w1
      Contact( "TRANSFER DB".BIT."MFG TO STORAGE-3 WITH INLINE FILTER PRES"."PBV-112 FILTER PRESS TO TRANSFER LINE" )
   END_RUNG wire#w2
   // the same network as SCL:
   "TRANSFER DB".OUTPUT."PBV-112 FILTER PRESS TO TRANSFER LINE" := "AlwaysTRUE" AND ("MODE SELECTION DB"."MODE BUFF" <> 0) AND ("TRANSFER DB".BIT."MFG TO STORAGE-1 WITH INLINE FILTER PRES"."PBV-112 FILTER PRESS TO TRANSFER LINE" OR "TRANSFER DB".BIT."MFG TO STORAGE-2 WITH INLINE FILTER PRES"."PBV-112 FILTER PRESS TO TRANSFER LINE" OR "TRANSFER DB".BIT."MFG TO STORAGE-3 WITH INLINE FILTER PRES"."PBV-112 FILTER PRESS TO TRANSFER LINE");
END_REGION

REGION Network 85: PAV-113 TANK OUTLET TO CIP DRAIN LINE
   RUNG wire#powerrail
      Contact( "AlwaysFALSE" )
      { S7_Templates := "SrcType := Int" } NE_Contact(in1 := "MODE SELECTION DB"."MODE BUFF", in2 := 0)
      Coil( "TRANSFER DB".OUTPUT."PAV-113 TANK OUTLET TO CIP DRAIN LINE" )
   END_RUNG
   // the same network as SCL:
   "TRANSFER DB".OUTPUT."PAV-113 TANK OUTLET TO CIP DRAIN LINE" := "AlwaysFALSE" AND ("MODE SELECTION DB"."MODE BUFF" <> 0);
END_REGION

REGION Network 86: PBV-114 TANK OUTLET TO INLINE HOMOGENIZER LINE
   RUNG wire#powerrail
      Contact( "AlwaysTRUE" )
      wire#w1
      { S7_Templates := "SrcType := Int" } NE_Contact(in1 := "MODE SELECTION DB"."MODE BUFF", in2 := 0)
      wire#w2
      Contact( "TRANSFER DB".BIT."MFG TO STORAGE-1 WITH INLINE HOMO"."PBV-114 TANK OUTLET TO INLINE HOMOGENIZER LINE" )
      wire#w3
      Coil( "TRANSFER DB".OUTPUT."PBV-114 TANK OUTLET TO INLINE HOMOGENIZER LINE" )
   END_RUNG
   RUNG wire#w2
      Contact( "TRANSFER DB".BIT."MFG TO STORAGE-1 WITH INLINE FILTER PRES"."PBV-114 TANK OUTLET TO INLINE HOMOGENIZER LINE" )
   END_RUNG wire#w3
   RUNG wire#w2
      Contact( "TRANSFER DB".BIT."MFG TO STORAGE-2 WITH INLINE HOMO"."PBV-114 TANK OUTLET TO INLINE HOMOGENIZER LINE" )
   END_RUNG wire#w3
   RUNG wire#w2
      Contact( "TRANSFER DB".BIT."MFG TO STORAGE-2 WITH INLINE FILTER PRES"."PBV-114 TANK OUTLET TO INLINE HOMOGENIZER LINE" )
   END_RUNG wire#w3
   RUNG wire#w2
      Contact( "TRANSFER DB".BIT."MFG TO STORAGE-3 WITH INLINE HOMO"."PBV-114 TANK OUTLET TO INLINE HOMOGENIZER LINE" )
   END_RUNG wire#w3
   RUNG wire#w2
      Contact( "TRANSFER DB".BIT."MFG TO STORAGE-3 WITH INLINE FILTER PRES"."PBV-114 TANK OUTLET TO INLINE HOMOGENIZER LINE" )
   END_RUNG wire#w3
   RUNG wire#w1
      { S7_Templates := "SrcType := Int" } EQ_Contact(in1 := "MODE SELECTION DB"."MODE BUFF", in2 := 2)
      { S7_Templates := "SrcType := Int" } EQ_Contact(in1 := "RECIRCULATION DB".MFG.BUFF, in2 := 2)
      I_Contact( "RECIRCULATION DB".MFG.PAUSE )
   END_RUNG wire#w3
   // the same network as SCL:
   "TRANSFER DB".OUTPUT."PBV-114 TANK OUTLET TO INLINE HOMOGENIZER LINE" := "AlwaysTRUE" AND ((("MODE SELECTION DB"."MODE BUFF" <> 0) AND ("TRANSFER DB".BIT."MFG TO STORAGE-1 WITH INLINE HOMO"."PBV-114 TANK OUTLET TO INLINE HOMOGENIZER LINE" OR "TRANSFER DB".BIT."MFG TO STORAGE-1 WITH INLINE FILTER PRES"."PBV-114 TANK OUTLET TO INLINE HOMOGENIZER LINE" OR "TRANSFER DB".BIT."MFG TO STORAGE-2 WITH INLINE HOMO"."PBV-114 TANK OUTLET TO INLINE HOMOGENIZER LINE" OR "TRANSFER DB".BIT."MFG TO STORAGE-2 WITH INLINE FILTER PRES"."PBV-114 TANK OUTLET TO INLINE HOMOGENIZER LINE" OR "TRANSFER DB".BIT."MFG TO STORAGE-3 WITH INLINE HOMO"."PBV-114 TANK OUTLET TO INLINE HOMOGENIZER LINE" OR "TRANSFER DB".BIT."MFG TO STORAGE-3 WITH INLINE FILTER PRES"."PBV-114 TANK OUTLET TO INLINE HOMOGENIZER LINE")) OR (("MODE SELECTION DB"."MODE BUFF" = 2) AND ("RECIRCULATION DB".MFG.BUFF = 2) AND NOT "RECIRCULATION DB".MFG.PAUSE));
END_REGION

REGION Network 87: PBV-115 MFG TO STORAGE – 1 TRANSFER LINE
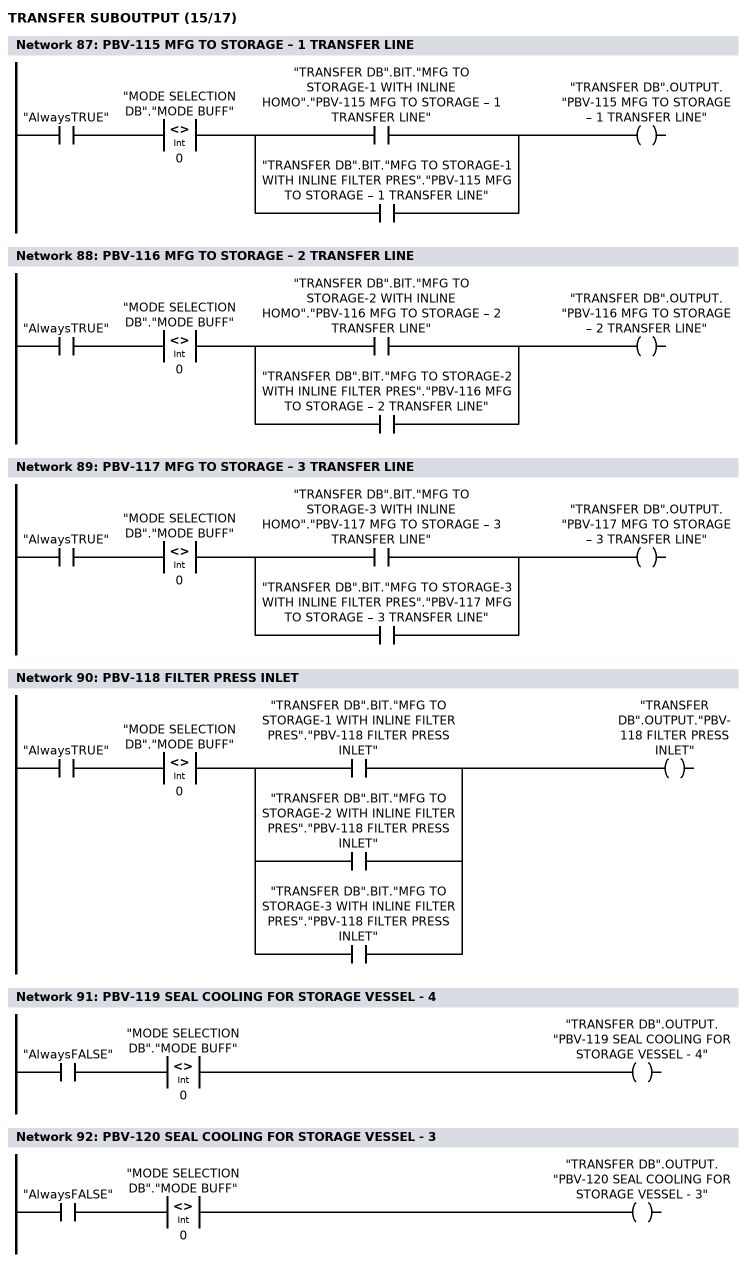
   RUNG wire#powerrail
      Contact( "AlwaysTRUE" )
      { S7_Templates := "SrcType := Int" } NE_Contact(in1 := "MODE SELECTION DB"."MODE BUFF", in2 := 0)
      wire#w1
      Contact( "TRANSFER DB".BIT."MFG TO STORAGE-1 WITH INLINE HOMO"."PBV-115 MFG TO STORAGE – 1 TRANSFER LINE" )
      wire#w2
      Coil( "TRANSFER DB".OUTPUT."PBV-115 MFG TO STORAGE – 1 TRANSFER LINE" )
   END_RUNG
   RUNG wire#w1
      Contact( "TRANSFER DB".BIT."MFG TO STORAGE-1 WITH INLINE FILTER PRES"."PBV-115 MFG TO STORAGE – 1 TRANSFER LINE" )
   END_RUNG wire#w2
   // the same network as SCL:
   "TRANSFER DB".OUTPUT."PBV-115 MFG TO STORAGE – 1 TRANSFER LINE" := "AlwaysTRUE" AND ("MODE SELECTION DB"."MODE BUFF" <> 0) AND ("TRANSFER DB".BIT."MFG TO STORAGE-1 WITH INLINE HOMO"."PBV-115 MFG TO STORAGE – 1 TRANSFER LINE" OR "TRANSFER DB".BIT."MFG TO STORAGE-1 WITH INLINE FILTER PRES"."PBV-115 MFG TO STORAGE – 1 TRANSFER LINE");
END_REGION

REGION Network 88: PBV-116 MFG TO STORAGE – 2 TRANSFER LINE
   RUNG wire#powerrail
      Contact( "AlwaysTRUE" )
      { S7_Templates := "SrcType := Int" } NE_Contact(in1 := "MODE SELECTION DB"."MODE BUFF", in2 := 0)
      wire#w1
      Contact( "TRANSFER DB".BIT."MFG TO STORAGE-2 WITH INLINE HOMO"."PBV-116 MFG TO STORAGE – 2 TRANSFER LINE" )
      wire#w2
      Coil( "TRANSFER DB".OUTPUT."PBV-116 MFG TO STORAGE – 2 TRANSFER LINE" )
   END_RUNG
   RUNG wire#w1
      Contact( "TRANSFER DB".BIT."MFG TO STORAGE-2 WITH INLINE FILTER PRES"."PBV-116 MFG TO STORAGE – 2 TRANSFER LINE" )
   END_RUNG wire#w2
   // the same network as SCL:
   "TRANSFER DB".OUTPUT."PBV-116 MFG TO STORAGE – 2 TRANSFER LINE" := "AlwaysTRUE" AND ("MODE SELECTION DB"."MODE BUFF" <> 0) AND ("TRANSFER DB".BIT."MFG TO STORAGE-2 WITH INLINE HOMO"."PBV-116 MFG TO STORAGE – 2 TRANSFER LINE" OR "TRANSFER DB".BIT."MFG TO STORAGE-2 WITH INLINE FILTER PRES"."PBV-116 MFG TO STORAGE – 2 TRANSFER LINE");
END_REGION

REGION Network 89: PBV-117 MFG TO STORAGE – 3 TRANSFER LINE
   RUNG wire#powerrail
      Contact( "AlwaysTRUE" )
      { S7_Templates := "SrcType := Int" } NE_Contact(in1 := "MODE SELECTION DB"."MODE BUFF", in2 := 0)
      wire#w1
      Contact( "TRANSFER DB".BIT."MFG TO STORAGE-3 WITH INLINE HOMO"."PBV-117 MFG TO STORAGE – 3 TRANSFER LINE" )
      wire#w2
      Coil( "TRANSFER DB".OUTPUT."PBV-117 MFG TO STORAGE – 3 TRANSFER LINE" )
   END_RUNG
   RUNG wire#w1
      Contact( "TRANSFER DB".BIT."MFG TO STORAGE-3 WITH INLINE FILTER PRES"."PBV-117 MFG TO STORAGE – 3 TRANSFER LINE" )
   END_RUNG wire#w2
   // the same network as SCL:
   "TRANSFER DB".OUTPUT."PBV-117 MFG TO STORAGE – 3 TRANSFER LINE" := "AlwaysTRUE" AND ("MODE SELECTION DB"."MODE BUFF" <> 0) AND ("TRANSFER DB".BIT."MFG TO STORAGE-3 WITH INLINE HOMO"."PBV-117 MFG TO STORAGE – 3 TRANSFER LINE" OR "TRANSFER DB".BIT."MFG TO STORAGE-3 WITH INLINE FILTER PRES"."PBV-117 MFG TO STORAGE – 3 TRANSFER LINE");
END_REGION

REGION Network 90: PBV-118 FILTER PRESS INLET
   RUNG wire#powerrail
      Contact( "AlwaysTRUE" )
      { S7_Templates := "SrcType := Int" } NE_Contact(in1 := "MODE SELECTION DB"."MODE BUFF", in2 := 0)
      wire#w1
      Contact( "TRANSFER DB".BIT."MFG TO STORAGE-1 WITH INLINE FILTER PRES"."PBV-118 FILTER PRESS INLET" )
      wire#w2
      Coil( "TRANSFER DB".OUTPUT."PBV-118 FILTER PRESS INLET" )
   END_RUNG
   RUNG wire#w1
      Contact( "TRANSFER DB".BIT."MFG TO STORAGE-2 WITH INLINE FILTER PRES"."PBV-118 FILTER PRESS INLET" )
   END_RUNG wire#w2
   RUNG wire#w1
      Contact( "TRANSFER DB".BIT."MFG TO STORAGE-3 WITH INLINE FILTER PRES"."PBV-118 FILTER PRESS INLET" )
   END_RUNG wire#w2
   // the same network as SCL:
   "TRANSFER DB".OUTPUT."PBV-118 FILTER PRESS INLET" := "AlwaysTRUE" AND ("MODE SELECTION DB"."MODE BUFF" <> 0) AND ("TRANSFER DB".BIT."MFG TO STORAGE-1 WITH INLINE FILTER PRES"."PBV-118 FILTER PRESS INLET" OR "TRANSFER DB".BIT."MFG TO STORAGE-2 WITH INLINE FILTER PRES"."PBV-118 FILTER PRESS INLET" OR "TRANSFER DB".BIT."MFG TO STORAGE-3 WITH INLINE FILTER PRES"."PBV-118 FILTER PRESS INLET");
END_REGION

REGION Network 91: PBV-119 SEAL COOLING FOR STORAGE VESSEL - 4
   RUNG wire#powerrail
      Contact( "AlwaysFALSE" )
      { S7_Templates := "SrcType := Int" } NE_Contact(in1 := "MODE SELECTION DB"."MODE BUFF", in2 := 0)
      Coil( "TRANSFER DB".OUTPUT."PBV-119 SEAL COOLING FOR STORAGE VESSEL - 4" )
   END_RUNG
   // the same network as SCL:
   "TRANSFER DB".OUTPUT."PBV-119 SEAL COOLING FOR STORAGE VESSEL - 4" := "AlwaysFALSE" AND ("MODE SELECTION DB"."MODE BUFF" <> 0);
END_REGION

REGION Network 92: PBV-120 SEAL COOLING FOR STORAGE VESSEL - 3
   RUNG wire#powerrail
      Contact( "AlwaysFALSE" )
      { S7_Templates := "SrcType := Int" } NE_Contact(in1 := "MODE SELECTION DB"."MODE BUFF", in2 := 0)
      Coil( "TRANSFER DB".OUTPUT."PBV-120 SEAL COOLING FOR STORAGE VESSEL - 3" )
   END_RUNG
   // the same network as SCL:
   "TRANSFER DB".OUTPUT."PBV-120 SEAL COOLING FOR STORAGE VESSEL - 3" := "AlwaysFALSE" AND ("MODE SELECTION DB"."MODE BUFF" <> 0);
END_REGION

REGION Network 93: PBV-121 SEAL COOLING FOR STORAGE VESSEL - 2
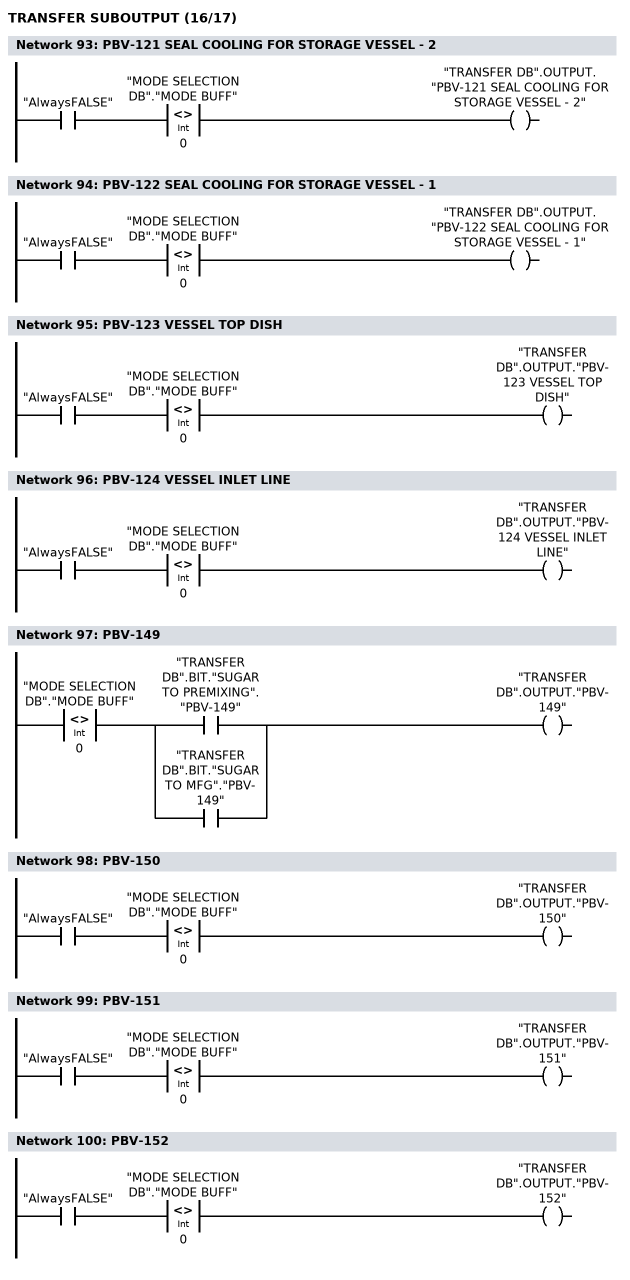
   RUNG wire#powerrail
      Contact( "AlwaysFALSE" )
      { S7_Templates := "SrcType := Int" } NE_Contact(in1 := "MODE SELECTION DB"."MODE BUFF", in2 := 0)
      Coil( "TRANSFER DB".OUTPUT."PBV-121 SEAL COOLING FOR STORAGE VESSEL - 2" )
   END_RUNG
   // the same network as SCL:
   "TRANSFER DB".OUTPUT."PBV-121 SEAL COOLING FOR STORAGE VESSEL - 2" := "AlwaysFALSE" AND ("MODE SELECTION DB"."MODE BUFF" <> 0);
END_REGION

REGION Network 94: PBV-122 SEAL COOLING FOR STORAGE VESSEL - 1
   RUNG wire#powerrail
      Contact( "AlwaysFALSE" )
      { S7_Templates := "SrcType := Int" } NE_Contact(in1 := "MODE SELECTION DB"."MODE BUFF", in2 := 0)
      Coil( "TRANSFER DB".OUTPUT."PBV-122 SEAL COOLING FOR STORAGE VESSEL - 1" )
   END_RUNG
   // the same network as SCL:
   "TRANSFER DB".OUTPUT."PBV-122 SEAL COOLING FOR STORAGE VESSEL - 1" := "AlwaysFALSE" AND ("MODE SELECTION DB"."MODE BUFF" <> 0);
END_REGION

REGION Network 95: PBV-123 VESSEL TOP DISH
   RUNG wire#powerrail
      Contact( "AlwaysFALSE" )
      { S7_Templates := "SrcType := Int" } NE_Contact(in1 := "MODE SELECTION DB"."MODE BUFF", in2 := 0)
      Coil( "TRANSFER DB".OUTPUT."PBV-123 VESSEL TOP DISH" )
   END_RUNG
   // the same network as SCL:
   "TRANSFER DB".OUTPUT."PBV-123 VESSEL TOP DISH" := "AlwaysFALSE" AND ("MODE SELECTION DB"."MODE BUFF" <> 0);
END_REGION

REGION Network 96: PBV-124 VESSEL INLET LINE
   RUNG wire#powerrail
      Contact( "AlwaysFALSE" )
      { S7_Templates := "SrcType := Int" } NE_Contact(in1 := "MODE SELECTION DB"."MODE BUFF", in2 := 0)
      Coil( "TRANSFER DB".OUTPUT."PBV-124 VESSEL INLET LINE" )
   END_RUNG
   // the same network as SCL:
   "TRANSFER DB".OUTPUT."PBV-124 VESSEL INLET LINE" := "AlwaysFALSE" AND ("MODE SELECTION DB"."MODE BUFF" <> 0);
END_REGION

REGION Network 97: PBV-149
   RUNG wire#powerrail
      { S7_Templates := "SrcType := Int" } NE_Contact(in1 := "MODE SELECTION DB"."MODE BUFF", in2 := 0)
      wire#w1
      Contact( "TRANSFER DB".BIT."SUGAR TO PREMIXING"."PBV-149" )
      wire#w2
      Coil( "TRANSFER DB".OUTPUT."PBV-149" )
   END_RUNG
   RUNG wire#w1
      Contact( "TRANSFER DB".BIT."SUGAR TO MFG"."PBV-149" )
   END_RUNG wire#w2
   // the same network as SCL:
   "TRANSFER DB".OUTPUT."PBV-149" := ("MODE SELECTION DB"."MODE BUFF" <> 0) AND ("TRANSFER DB".BIT."SUGAR TO PREMIXING"."PBV-149" OR "TRANSFER DB".BIT."SUGAR TO MFG"."PBV-149");
END_REGION

REGION Network 98: PBV-150
   RUNG wire#powerrail
      Contact( "AlwaysFALSE" )
      { S7_Templates := "SrcType := Int" } NE_Contact(in1 := "MODE SELECTION DB"."MODE BUFF", in2 := 0)
      Coil( "TRANSFER DB".OUTPUT."PBV-150" )
   END_RUNG
   // the same network as SCL:
   "TRANSFER DB".OUTPUT."PBV-150" := "AlwaysFALSE" AND ("MODE SELECTION DB"."MODE BUFF" <> 0);
END_REGION

REGION Network 99: PBV-151
   RUNG wire#powerrail
      Contact( "AlwaysFALSE" )
      { S7_Templates := "SrcType := Int" } NE_Contact(in1 := "MODE SELECTION DB"."MODE BUFF", in2 := 0)
      Coil( "TRANSFER DB".OUTPUT."PBV-151" )
   END_RUNG
   // the same network as SCL:
   "TRANSFER DB".OUTPUT."PBV-151" := "AlwaysFALSE" AND ("MODE SELECTION DB"."MODE BUFF" <> 0);
END_REGION

REGION Network 100: PBV-152
   RUNG wire#powerrail
      Contact( "AlwaysFALSE" )
      { S7_Templates := "SrcType := Int" } NE_Contact(in1 := "MODE SELECTION DB"."MODE BUFF", in2 := 0)
      Coil( "TRANSFER DB".OUTPUT."PBV-152" )
   END_RUNG
   // the same network as SCL:
   "TRANSFER DB".OUTPUT."PBV-152" := "AlwaysFALSE" AND ("MODE SELECTION DB"."MODE BUFF" <> 0);
END_REGION

REGION Network 101: PBV-153
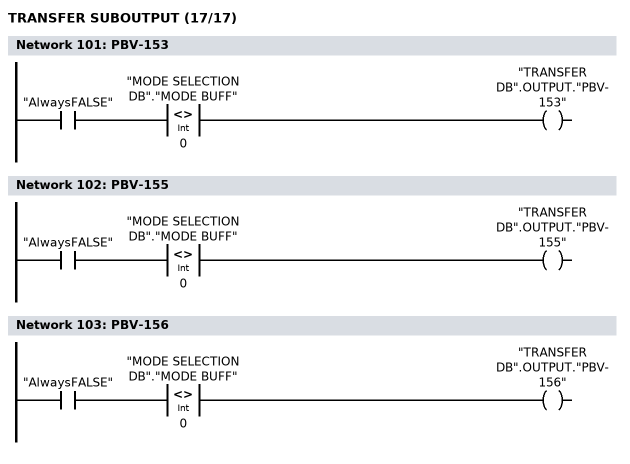
   RUNG wire#powerrail
      Contact( "AlwaysFALSE" )
      { S7_Templates := "SrcType := Int" } NE_Contact(in1 := "MODE SELECTION DB"."MODE BUFF", in2 := 0)
      Coil( "TRANSFER DB".OUTPUT."PBV-153" )
   END_RUNG
   // the same network as SCL:
   "TRANSFER DB".OUTPUT."PBV-153" := "AlwaysFALSE" AND ("MODE SELECTION DB"."MODE BUFF" <> 0);
END_REGION

REGION Network 102: PBV-155
   RUNG wire#powerrail
      Contact( "AlwaysFALSE" )
      { S7_Templates := "SrcType := Int" } NE_Contact(in1 := "MODE SELECTION DB"."MODE BUFF", in2 := 0)
      Coil( "TRANSFER DB".OUTPUT."PBV-155" )
   END_RUNG
   // the same network as SCL:
   "TRANSFER DB".OUTPUT."PBV-155" := "AlwaysFALSE" AND ("MODE SELECTION DB"."MODE BUFF" <> 0);
END_REGION

REGION Network 103: PBV-156
   RUNG wire#powerrail
      Contact( "AlwaysFALSE" )
      { S7_Templates := "SrcType := Int" } NE_Contact(in1 := "MODE SELECTION DB"."MODE BUFF", in2 := 0)
      Coil( "TRANSFER DB".OUTPUT."PBV-156" )
   END_RUNG
   // the same network as SCL:
   "TRANSFER DB".OUTPUT."PBV-156" := "AlwaysFALSE" AND ("MODE SELECTION DB"."MODE BUFF" <> 0);
END_REGION
END_FUNCTION
